LIN {X 0,Y 467.685,Z 587.224,A -85,B 0,C 180,E1 -7551.357,E2 -7551.357} C_VEL
LIN {X 0,Y 467.743,Z 587.223,A -85,B 0,C 180,E1 -7553.963,E2 -7553.963} C_VEL
LIN {X 0,Y 467.864,Z 587.201,A -85,B 0,C 180,E1 -7557.417,E2 -7557.417} C_VEL
LIN {X 0,Y 467.888,Z 587.204,A -85,B 0,C 180,E1 -7560,E2 -7560} C_VEL
LIN {X 0,Y 467.864,Z 587.204,A -85,B 0,C 180,E1 -7562.583,E2 -7562.583} C_VEL
LIN {X 0,Y 467.748,Z 587.22,A -85,B 0,C 180,E1 -7566.037,E2 -7566.037} C_VEL
LIN {X 0,Y 467.686,Z 587.227,A -85,B 0,C 180,E1 -7568.643,E2 -7568.643} C_VEL
LIN {X 0,Y 467.662,Z 587.231,A -85,B 0,C 180,E1 -7572.145,E2 -7572.145} C_VEL
LIN {X 0,Y 467.645,Z 587.228,A -85,B 0,C 180,E1 -7575.695,E2 -7575.695} C_VEL
LIN {X 0,Y 467.619,Z 587.237,A -85,B 0,C 180,E1 -7578.763,E2 -7578.763} C_VEL
LIN {X 0,Y 467.586,Z 587.236,A -85,B 0,C 180,E1 -7581.268,E2 -7581.268} C_VEL
LIN {X 0,Y 467.576,Z 587.237,A -85,B 0,C 180,E1 -7583.943,E2 -7583.943} C_VEL
LIN {X 0,Y 467.622,Z 587.238,A -85,B 0,C 180,E1 -7586.8,E2 -7586.8} C_VEL
LIN {X 0,Y 467.56,Z 587.238,A -85,B 0,C 180,E1 -7589.738,E2 -7589.738} C_VEL
LIN {X 0,Y 467.589,Z 587.243,A -85,B 0,C 180,E1 -7592.758,E2 -7592.758} C_VEL
LIN {X 0,Y 467.559,Z 587.238,A -85,B 0,C 180,E1 -7595.889,E2 -7595.889} C_VEL
LIN {X 0,Y 467.581,Z 587.241,A -85,B 0,C 180,E1 -7599.145,E2 -7599.145} C_VEL
LIN {X 0,Y 467.592,Z 587.238,A -85,B 0,C 180,E1 -7602.567,E2 -7602.567} C_VEL
LIN {X 0,Y 467.576,Z 587.245,A -85,B 0,C 180,E1 -7605.053,E2 -7605.053} C_VEL
LIN {X 0,Y 467.594,Z 587.238,A -85,B 0,C 180,E1 -7607.44,E2 -7607.44} C_VEL
LIN {X 0,Y 467.588,Z 587.24,A -85,B 0,C 180,E1 -7610.855,E2 -7610.855} C_VEL
LIN {X 0,Y 467.565,Z 587.238,A -85,B 0,C 180,E1 -7614.26,E2 -7614.26} C_VEL
LIN {X 0,Y 467.587,Z 587.243,A -85,B 0,C 180,E1 -7617.32,E2 -7617.32} C_VEL
LIN {X 0,Y 467.574,Z 587.241,A -85,B 0,C 180,E1 -7620.667,E2 -7620.667} C_VEL
LIN {X 0,Y 467.688,Z 587.373,A -85,B 0,C 180,E1 -7622.729,E2 -7622.729} C_VEL
LIN {X 0,Y 470.217,Z 599.912,A -85,B 0,C 180,E1 -7625.024,E2 -7625.024} C_VEL
LIN {X 0,Y 470.285,Z 605.726,A -85,B 0,C 180,E1 -7626.017,E2 -7626.017} C_VEL
LIN {X 0,Y 469.404,Z 623.346,A -85,B 0,C 180,E1 -7628.94,E2 -7628.94} C_VEL
LIN {X 0,Y 468.7,Z 641.213,A -85,B 0,C 180,E1 -7631.871,E2 -7631.871} C_VEL
LIN {X 0,Y 468.432,Z 648.08,A -85,B 0,C 180,E1 -7632.987,E2 -7632.987} C_VEL
LIN {X 0,Y 471.155,Z 668.22,A -85,B 0,C 180,E1 -7633.412,E2 -7633.412} C_VEL
LIN {X 0,Y 470.414,Z 757.203,A -85,B 0,C 180,E1 -7634.843,E2 -7634.843} C_VEL
LIN {X 0,Y 469.976,Z 771.033,A -85,B 0,C 180,E1 -7635.244,E2 -7635.244} C_VEL
LIN {X 0,Y 469.566,Z 784.014,A -85,B 0,C 180,E1 -7635.812,E2 -7635.812} C_VEL
LIN {X 0,Y 469.023,Z 796.625,A -85,B 0,C 180,E1 -7636.569,E2 -7636.569} C_VEL
LIN {X 0,Y 468.588,Z 807.32,A -85,B 0,C 180,E1 -7637.39,E2 -7637.39} C_VEL
LIN {X 0,Y 468.191,Z 817.018,A -85,B 0,C 180,E1 -7638.307,E2 -7638.307} C_VEL
LIN {X 0,Y 467.667,Z 826.375,A -85,B 0,C 180,E1 -7639.391,E2 -7639.391} C_VEL
LIN {X 0,Y 467.284,Z 835.456,A -85,B 0,C 180,E1 -7640.695,E2 -7640.695} C_VEL
LIN {X 0,Y 467.022,Z 842.773,A -85,B 0,C 180,E1 -7641.998,E2 -7641.998} C_VEL
LIN {X 0,Y 466.855,Z 847.713,A -85,B 0,C 180,E1 -7643.082,E2 -7643.082} C_VEL
LIN {X 0,Y 466.787,Z 852.513,A -85,B 0,C 180,E1 -7644.383,E2 -7644.383} C_VEL
LIN {X 0,Y 466.666,Z 856.175,A -85,B 0,C 180,E1 -7645.681,E2 -7645.681} C_VEL
LIN {X 0,Y 466.728,Z 858.07,A -85,B 0,C 180,E1 -7646.546,E2 -7646.546} C_VEL
LIN {X 0,Y 466.7,Z 859.486,A -85,B 0,C 180,E1 -7647.41,E2 -7647.41} C_VEL
LIN {X 0,Y 466.693,Z 860.49,A -85,B 0,C 180,E1 -7648.273,E2 -7648.273} C_VEL
LIN {X 0,Y 466.598,Z 861.304,A -85,B 0,C 180,E1 -7649.999,E2 -7649.999} C_VEL
LIN {X 0,Y 466.62,Z 861.075,A -85,B 0,C 180,E1 -7650.862,E2 -7650.862} C_VEL
LIN {X 0,Y 466.694,Z 860.447,A -85,B 0,C 180,E1 -7651.725,E2 -7651.725} C_VEL
LIN {X 0,Y 466.71,Z 859.42,A -85,B 0,C 180,E1 -7652.588,E2 -7652.588} C_VEL
LIN {X 0,Y 466.728,Z 857.982,A -85,B 0,C 180,E1 -7653.452,E2 -7653.452} C_VEL
LIN {X 0,Y 466.7,Z 854.965,A -85,B 0,C 180,E1 -7654.75,E2 -7654.75} C_VEL
LIN {X 0,Y 466.768,Z 850.892,A -85,B 0,C 180,E1 -7656.049,E2 -7656.049} C_VEL
LIN {X 0,Y 466.928,Z 844.629,A -85,B 0,C 180,E1 -7657.567,E2 -7657.567} C_VEL
LIN {X 0,Y 467.165,Z 837.801,A -85,B 0,C 180,E1 -7658.869,E2 -7658.869} C_VEL
LIN {X 0,Y 467.497,Z 829.332,A -85,B 0,C 180,E1 -7660.173,E2 -7660.173} C_VEL
LIN {X 0,Y 467.921,Z 820.622,A -85,B 0,C 180,E1 -7661.259,E2 -7661.259} C_VEL
LIN {X 0,Y 468.377,Z 810.405,A -85,B 0,C 180,E1 -7662.298,E2 -7662.298} C_VEL
LIN {X 0,Y 468.893,Z 799.253,A -85,B 0,C 180,E1 -7663.212,E2 -7663.212} C_VEL
LIN {X 0,Y 469.367,Z 787.483,A -85,B 0,C 180,E1 -7663.971,E2 -7663.971} C_VEL
LIN {X 0,Y 469.795,Z 775.278,A -85,B 0,C 180,E1 -7664.566,E2 -7664.566} C_VEL
LIN {X 0,Y 470.222,Z 762.96,A -85,B 0,C 180,E1 -7664.995,E2 -7664.995} C_VEL
LIN {X 0,Y 470.484,Z 749.275,A -85,B 0,C 180,E1 -7665.291,E2 -7665.291} C_VEL
LIN {X 0,Y 471.087,Z 666.51,A -85,B 0,C 180,E1 -7666.607,E2 -7666.607} C_VEL
LIN {X 0,Y 468.342,Z 647.034,A -85,B 0,C 180,E1 -7667.056,E2 -7667.056} C_VEL
LIN {X 0,Y 469.089,Z 627.979,A -85,B 0,C 180,E1 -7670.156,E2 -7670.156} C_VEL
LIN {X 0,Y 469.848,Z 610.048,A -85,B 0,C 180,E1 -7673.118,E2 -7673.118} C_VEL
LIN {X 0,Y 470.271,Z 600.433,A -85,B 0,C 180,E1 -7674.735,E2 -7674.735} C_VEL
LIN {X 0,Y 467.669,Z 587.232,A -85,B 0,C 180,E1 -7677.189,E2 -7677.189} C_VEL
LIN {X 0,Y 467.568,Z 587.248,A -85,B 0,C 180,E1 -7680.733,E2 -7680.733} C_VEL
LIN {X 0,Y 467.584,Z 587.24,A -85,B 0,C 180,E1 -7683.787,E2 -7683.787} C_VEL
LIN {X 0,Y 467.548,Z 587.244,A -85,B 0,C 180,E1 -7687.186,E2 -7687.186} C_VEL
LIN {X 0,Y 467.591,Z 587.243,A -85,B 0,C 180,E1 -7690.262,E2 -7690.262} C_VEL
LIN {X 0,Y 467.582,Z 587.245,A -85,B 0,C 180,E1 -7692.566,E2 -7692.566} C_VEL
LIN {X 0,Y 467.57,Z 587.245,A -85,B 0,C 180,E1 -7696.175,E2 -7696.175} C_VEL
LIN {X 0,Y 467.584,Z 587.242,A -85,B 0,C 180,E1 -7698.721,E2 -7698.721} C_VEL
LIN {X 0,Y 467.573,Z 587.238,A -85,B 0,C 180,E1 -7701.405,E2 -7701.405} C_VEL
LIN {X 0,Y 467.557,Z 587.244,A -85,B 0,C 180,E1 -7704.259,E2 -7704.259} C_VEL
LIN {X 0,Y 467.576,Z 587.237,A -85,B 0,C 180,E1 -7707.32,E2 -7707.32} C_VEL
LIN {X 0,Y 467.572,Z 587.24,A -85,B 0,C 180,E1 -7710.665,E2 -7710.665} C_VEL
LIN {X 0,Y 467.62,Z 587.231,A -85,B 0,C 180,E1 -7713.2,E2 -7713.2} C_VEL
LIN {X 0,Y 467.585,Z 587.24,A -85,B 0,C 180,E1 -7716.467,E2 -7716.467} C_VEL
LIN {X 0,Y 467.616,Z 587.232,A -85,B 0,C 180,E1 -7719.777,E2 -7719.777} C_VEL
LIN {X 0,Y 467.601,Z 587.239,A -85,B 0,C 180,E1 -7722.506,E2 -7722.506} C_VEL
LIN {X 0,Y 467.598,Z 587.234,A -85,B 0,C 180,E1 -7725.196,E2 -7725.196} C_VEL
LIN {X 0,Y 467.674,Z 587.227,A -85,B 0,C 180,E1 -7727.855,E2 -7727.855} C_VEL
LIN {X 0,Y 467.674,Z 587.226,A -85,B 0,C 180,E1 -7731.357,E2 -7731.357} C_VEL
LIN {X 0,Y 467.735,Z 587.222,A -85,B 0,C 180,E1 -7733.962,E2 -7733.962} C_VEL
LIN {X 0,Y 467.852,Z 587.204,A -85,B 0,C 180,E1 -7737.417,E2 -7737.417} C_VEL
LIN {X 0,Y 467.874,Z 587.206,A -85,B 0,C 180,E1 -7740,E2 -7740} C_VEL
LIN {X 0,Y 467.852,Z 587.209,A -85,B 0,C 180,E1 -7742.583,E2 -7742.583} C_VEL
LIN {X 0,Y 467.746,Z 587.224,A -85,B 0,C 180,E1 -7746.037,E2 -7746.037} C_VEL
LIN {X 0,Y 467.674,Z 587.231,A -85,B 0,C 180,E1 -7748.643,E2 -7748.643} C_VEL
LIN {X 0,Y 467.675,Z 587.235,A -85,B 0,C 180,E1 -7752.145,E2 -7752.145} C_VEL
LIN {X 0,Y 467.661,Z 587.255,A -85,B 0,C 180,E1 -7755.359,E2 -7755.359} C_VEL
LIN {X 0,Y 468.623,Z 593.879,A -85,B 0,C 180,E1 -7757.004,E2 -7757.004} C_VEL
LIN {X 0,Y 468.56,Z 598.288,A -85,B 0,C 180,E1 -7758.049,E2 -7758.049} C_VEL
LIN {X 0,Y 471.347,Z 611.243,A -85,B 0,C 180,E1 -7758.388,E2 -7758.388} C_VEL
LIN {X 0,Y 470.527,Z 704.015,A -85,B 0,C 180,E1 -7759.891,E2 -7759.891} C_VEL
LIN {X 0,Y 470.243,Z 717.329,A -85,B 0,C 180,E1 -7760.276,E2 -7760.276} C_VEL
LIN {X 0,Y 469.916,Z 729.669,A -85,B 0,C 180,E1 -7760.806,E2 -7760.806} C_VEL
LIN {X 0,Y 469.564,Z 741.214,A -85,B 0,C 180,E1 -7761.474,E2 -7761.474} C_VEL
LIN {X 0,Y 469.048,Z 752.847,A -85,B 0,C 180,E1 -7762.346,E2 -7762.346} C_VEL
LIN {X 0,Y 468.564,Z 762.941,A -85,B 0,C 180,E1 -7763.293,E2 -7763.293} C_VEL
LIN {X 0,Y 468.102,Z 772.4,A -85,B 0,C 180,E1 -7764.386,E2 -7764.386} C_VEL
LIN {X 0,Y 467.651,Z 780.999,A -85,B 0,C 180,E1 -7765.621,E2 -7765.621} C_VEL
LIN {X 0,Y 467.375,Z 787.765,A -85,B 0,C 180,E1 -7766.815,E2 -7766.815} C_VEL
LIN {X 0,Y 467.121,Z 794.44,A -85,B 0,C 180,E1 -7768.29,E2 -7768.29} C_VEL
LIN {X 0,Y 466.865,Z 799.568,A -85,B 0,C 180,E1 -7769.786,E2 -7769.786} C_VEL
LIN {X 0,Y 466.807,Z 802.45,A -85,B 0,C 180,E1 -7770.892,E2 -7770.892} C_VEL
LIN {X 0,Y 466.639,Z 805.331,A -85,B 0,C 180,E1 -7772.5,E2 -7772.5} C_VEL
LIN {X 0,Y 466.576,Z 806.772,A -85,B 0,C 180,E1 -7774.061,E2 -7774.061} C_VEL
LIN {X 0,Y 466.56,Z 806.938,A -85,B 0,C 180,E1 -7775.57,E2 -7775.57} C_VEL
LIN {X 0,Y 466.592,Z 805.927,A -85,B 0,C 180,E1 -7777.049,E2 -7777.049} C_VEL
LIN {X 0,Y 466.696,Z 803.852,A -85,B 0,C 180,E1 -7778.459,E2 -7778.459} C_VEL
LIN {X 0,Y 466.821,Z 800.709,A -85,B 0,C 180,E1 -7779.845,E2 -7779.845} C_VEL
LIN {X 0,Y 467.007,Z 795.499,A -85,B 0,C 180,E1 -7781.465,E2 -7781.465} C_VEL
LIN {X 0,Y 467.231,Z 789.418,A -85,B 0,C 180,E1 -7782.894,E2 -7782.894} C_VEL
LIN {X 0,Y 467.618,Z 781.516,A -85,B 0,C 180,E1 -7784.335,E2 -7784.335} C_VEL
LIN {X 0,Y 468.027,Z 773.201,A -85,B 0,C 180,E1 -7785.55,E2 -7785.55} C_VEL
LIN {X 0,Y 468.454,Z 764.065,A -85,B 0,C 180,E1 -7786.639,E2 -7786.639} C_VEL
LIN {X 0,Y 468.921,Z 754.232,A -85,B 0,C 180,E1 -7787.591,E2 -7787.591} C_VEL
LIN {X 0,Y 469.398,Z 742.869,A -85,B 0,C 180,E1 -7788.471,E2 -7788.471} C_VEL
LIN {X 0,Y 469.882,Z 730.838,A -85,B 0,C 180,E1 -7789.197,E2 -7789.197} C_VEL
LIN {X 0,Y 470.193,Z 717.902,A -85,B 0,C 180,E1 -7789.774,E2 -7789.774} C_VEL
LIN {X 0,Y 470.298,Z 712.356,A -85,B 0,C 180,E1 -7789.964,E2 -7789.964} C_VEL
LIN {X 0,Y 469.848,Z 706.643,A -85,B 0,C 180,E1 -7790.143,E2 -7790.143} C_VEL
LIN {X 0,Y 464.422,Z 688.031,A -85,B 0,C 180,E1 -7790.669,E2 -7790.669} C_VEL
LIN {X 0,Y 463.83,Z 682.219,A -85,B 0,C 180,E1 -7790.78,E2 -7790.78} C_VEL
LIN {X 0,Y 464.42,Z 611.549,A -85,B 0,C 180,E1 -7791.929,E2 -7791.929} C_VEL
LIN {X 0,Y 461.453,Z 597.515,A -85,B 0,C 180,E1 -7792.301,E2 -7792.301} C_VEL
LIN {X 0,Y 461.33,Z 592.208,A -85,B 0,C 180,E1 -7793.551,E2 -7793.551} C_VEL
LIN {X 0,Y 460.592,Z 588.114,A -85,B 0,C 180,E1 -7794.563,E2 -7794.563} C_VEL
LIN {X 0,Y 460.528,Z 588.121,A -85,B 0,C 180,E1 -7797.717,E2 -7797.717} C_VEL
LIN {X 0,Y 460.536,Z 588.114,A -85,B 0,C 180,E1 -7800.77,E2 -7800.77} C_VEL
LIN {X 0,Y 460.56,Z 588.114,A -85,B 0,C 180,E1 -7803.736,E2 -7803.736} C_VEL
LIN {X 0,Y 460.544,Z 588.115,A -85,B 0,C 180,E1 -7806.625,E2 -7806.625} C_VEL
LIN {X 0,Y 460.551,Z 588.112,A -85,B 0,C 180,E1 -7809.454,E2 -7809.454} C_VEL
LIN {X 0,Y 460.559,Z 588.119,A -85,B 0,C 180,E1 -7812.231,E2 -7812.231} C_VEL
LIN {X 0,Y 460.565,Z 588.111,A -85,B 0,C 180,E1 -7814.966,E2 -7814.966} C_VEL
LIN {X 0,Y 460.63,Z 588.103,A -85,B 0,C 180,E1 -7817.667,E2 -7817.667} C_VEL
LIN {X 0,Y 460.629,Z 588.102,A -85,B 0,C 180,E1 -7821.225,E2 -7821.225} C_VEL
LIN {X 0,Y 460.71,Z 588.093,A -85,B 0,C 180,E1 -7823.871,E2 -7823.871} C_VEL
LIN {X 0,Y 460.826,Z 588.077,A -85,B 0,C 180,E1 -7827.379,E2 -7827.379} C_VEL
LIN {X 0,Y 460.854,Z 588.076,A -85,B 0,C 180,E1 -7830.001,E2 -7830.001} C_VEL
LIN {X 0,Y 460.827,Z 588.086,A -85,B 0,C 180,E1 -7832.623,E2 -7832.623} C_VEL
LIN {X 0,Y 460.712,Z 588.093,A -85,B 0,C 180,E1 -7836.131,E2 -7836.131} C_VEL
LIN {X 0,Y 460.632,Z 588.109,A -85,B 0,C 180,E1 -7838.777,E2 -7838.777} C_VEL
LIN {X 0,Y 460.616,Z 588.108,A -85,B 0,C 180,E1 -7842.446,E2 -7842.446} C_VEL
LIN {X 0,Y 460.603,Z 588.105,A -85,B 0,C 180,E1 -7845.998,E2 -7845.998} C_VEL
LIN {X 0,Y 460.574,Z 588.117,A -85,B 0,C 180,E1 -7848.903,E2 -7848.903} C_VEL
LIN {X 0,Y 460.519,Z 588.117,A -85,B 0,C 180,E1 -7851.486,E2 -7851.486} C_VEL
LIN {X 0,Y 460.545,Z 588.113,A -85,B 0,C 180,E1 -7854.333,E2 -7854.333} C_VEL
LIN {X 0,Y 460.577,Z 588.114,A -85,B 0,C 180,E1 -7857.244,E2 -7857.244} C_VEL
LIN {X 0,Y 460.514,Z 588.116,A -85,B 0,C 180,E1 -7860.241,E2 -7860.241} C_VEL
LIN {X 0,Y 460.533,Z 588.12,A -85,B 0,C 180,E1 -7863.325,E2 -7863.325} C_VEL
LIN {X 0,Y 460.481,Z 588.121,A -85,B 0,C 180,E1 -7866.53,E2 -7866.53} C_VEL
LIN {X 0,Y 460.536,Z 588.115,A -85,B 0,C 180,E1 -7869.863,E2 -7869.863} C_VEL
LIN {X 0,Y 460.517,Z 588.119,A -85,B 0,C 180,E1 -7872.901,E2 -7872.901} C_VEL
LIN {X 0,Y 460.513,Z 588.119,A -85,B 0,C 180,E1 -7875.831,E2 -7875.831} C_VEL
LIN {X 0,Y 460.535,Z 588.116,A -85,B 0,C 180,E1 -7878.989,E2 -7878.989} C_VEL
LIN {X 0,Y 460.523,Z 588.121,A -85,B 0,C 180,E1 -7881.267,E2 -7881.267} C_VEL
LIN {X 0,Y 460.515,Z 588.116,A -85,B 0,C 180,E1 -7884.555,E2 -7884.555} C_VEL
LIN {X 0,Y 460.536,Z 588.12,A -85,B 0,C 180,E1 -7887.716,E2 -7887.716} C_VEL
LIN {X 0,Y 460.544,Z 588.112,A -85,B 0,C 180,E1 -7890.769,E2 -7890.769} C_VEL
LIN {X 0,Y 460.561,Z 588.119,A -85,B 0,C 180,E1 -7893.735,E2 -7893.735} C_VEL
LIN {X 0,Y 460.549,Z 588.112,A -85,B 0,C 180,E1 -7896.624,E2 -7896.624} C_VEL
LIN {X 0,Y 460.556,Z 588.115,A -85,B 0,C 180,E1 -7899.453,E2 -7899.453} C_VEL
LIN {X 0,Y 460.555,Z 588.115,A -85,B 0,C 180,E1 -7902.23,E2 -7902.23} C_VEL
LIN {X 0,Y 460.57,Z 588.109,A -85,B 0,C 180,E1 -7904.965,E2 -7904.965} C_VEL
LIN {X 0,Y 460.615,Z 588.105,A -85,B 0,C 180,E1 -7908.559,E2 -7908.559} C_VEL
LIN {X 0,Y 460.701,Z 588.101,A -85,B 0,C 180,E1 -7912.109,E2 -7912.109} C_VEL
LIN {X 0,Y 460.7,Z 588.094,A -85,B 0,C 180,E1 -7914.748,E2 -7914.748} C_VEL
LIN {X 0,Y 460.805,Z 588.08,A -85,B 0,C 180,E1 -7917.378,E2 -7917.378} C_VEL
LIN {X 0,Y 460.858,Z 588.079,A -85,B 0,C 180,E1 -7920,E2 -7920} C_VEL
LIN {X 0,Y 460.805,Z 588.083,A -85,B 0,C 180,E1 -7922.623,E2 -7922.623} C_VEL
LIN {X 0,Y 460.714,Z 588.097,A -85,B 0,C 180,E1 -7926.13,E2 -7926.13} C_VEL
LIN {X 0,Y 460.633,Z 588.104,A -85,B 0,C 180,E1 -7928.776,E2 -7928.776} C_VEL
LIN {X 0,Y 460.619,Z 588.112,A -85,B 0,C 180,E1 -7932.445,E2 -7932.445} C_VEL
LIN {X 0,Y 460.606,Z 588.107,A -85,B 0,C 180,E1 -7935.997,E2 -7935.997} C_VEL
LIN {X 0,Y 460.574,Z 588.109,A -85,B 0,C 180,E1 -7939.615,E2 -7939.615} C_VEL
LIN {X 0,Y 460.517,Z 588.122,A -85,B 0,C 180,E1 -7942.429,E2 -7942.429} C_VEL
LIN {X 0,Y 460.563,Z 588.11,A -85,B 0,C 180,E1 -7945.799,E2 -7945.799} C_VEL
LIN {X 0,Y 460.558,Z 588.113,A -85,B 0,C 180,E1 -7948.233,E2 -7948.233} C_VEL
LIN {X 0,Y 460.526,Z 588.117,A -85,B 0,C 180,E1 -7951.283,E2 -7951.283} C_VEL
LIN {X 0,Y 460.538,Z 588.117,A -85,B 0,C 180,E1 -7954.505,E2 -7954.505} C_VEL
LIN {X 0,Y 460.507,Z 588.118,A -85,B 0,C 180,E1 -7957.623,E2 -7957.623} C_VEL
LIN {X 0,Y 460.544,Z 588.113,A -85,B 0,C 180,E1 -7960.269,E2 -7960.269} C_VEL
LIN {X 0,Y 460.506,Z 588.12,A -85,B 0,C 180,E1 -7963.375,E2 -7963.375} C_VEL
LIN {X 0,Y 460.506,Z 588.12,A -85,B 0,C 180,E1 -7966.624,E2 -7966.624} C_VEL
LIN {X 0,Y 460.547,Z 588.113,A -85,B 0,C 180,E1 -7969.73,E2 -7969.73} C_VEL
LIN {X 0,Y 460.505,Z 588.119,A -85,B 0,C 180,E1 -7972.523,E2 -7972.523} C_VEL
LIN {X 0,Y 460.552,Z 588.117,A -85,B 0,C 180,E1 -7975.623,E2 -7975.623} C_VEL
LIN {X 0,Y 460.542,Z 588.117,A -85,B 0,C 180,E1 -7978.744,E2 -7978.744} C_VEL
LIN {X 0,Y 460.586,Z 588.113,A -85,B 0,C 180,E1 -7982.253,E2 -7982.253} C_VEL
LIN {X 0,Y 460.625,Z 588.289,A -85,B 0,C 180,E1 -7982.51,E2 -7982.51} C_VEL
LIN {X 0,Y 463.403,Z 601.997,A -85,B 0,C 180,E1 -7985.057,E2 -7985.057} C_VEL
LIN {X 0,Y 463.036,Z 613.34,A -85,B 0,C 180,E1 -7986.993,E2 -7986.993} C_VEL
LIN {X 0,Y 462.049,Z 633.966,A -85,B 0,C 180,E1 -7990.449,E2 -7990.449} C_VEL
LIN {X 0,Y 461.432,Z 647.712,A -85,B 0,C 180,E1 -7992.723,E2 -7992.723} C_VEL
LIN {X 0,Y 464.321,Z 668.327,A -85,B 0,C 180,E1 -7993.177,E2 -7993.177} C_VEL
LIN {X 0,Y 463.52,Z 757.447,A -85,B 0,C 180,E1 -7994.64,E2 -7994.64} C_VEL
LIN {X 0,Y 463.053,Z 771.055,A -85,B 0,C 180,E1 -7995.047,E2 -7995.047} C_VEL
LIN {X 0,Y 462.656,Z 783.387,A -85,B 0,C 180,E1 -7995.596,E2 -7995.596} C_VEL
LIN {X 0,Y 462.086,Z 796.048,A -85,B 0,C 180,E1 -7996.364,E2 -7996.364} C_VEL
LIN {X 0,Y 461.58,Z 807.608,A -85,B 0,C 180,E1 -7997.267,E2 -7997.267} C_VEL
LIN {X 0,Y 461.138,Z 817.528,A -85,B 0,C 180,E1 -7998.237,E2 -7998.237} C_VEL
LIN {X 0,Y 460.551,Z 827.532,A -85,B 0,C 180,E1 -7999.448,E2 -7999.448} C_VEL
LIN {X 0,Y 460.192,Z 836.353,A -85,B 0,C 180,E1 -8000.772,E2 -8000.772} C_VEL
LIN {X 0,Y 459.899,Z 843.382,A -85,B 0,C 180,E1 -8002.094,E2 -8002.094} C_VEL
LIN {X 0,Y 459.715,Z 849.579,A -85,B 0,C 180,E1 -8003.568,E2 -8003.568} C_VEL
LIN {X 0,Y 459.631,Z 854.675,A -85,B 0,C 180,E1 -8005.175,E2 -8005.175} C_VEL
LIN {X 0,Y 459.625,Z 857.654,A -85,B 0,C 180,E1 -8006.493,E2 -8006.493} C_VEL
LIN {X 0,Y 459.621,Z 859.074,A -85,B 0,C 180,E1 -8007.37,E2 -8007.37} C_VEL
LIN {X 0,Y 459.63,Z 860.08,A -85,B 0,C 180,E1 -8008.247,E2 -8008.247} C_VEL
LIN {X 0,Y 459.53,Z 860.893,A -85,B 0,C 180,E1 -8009.999,E2 -8009.999} C_VEL
LIN {X 0,Y 459.553,Z 860.662,A -85,B 0,C 180,E1 -8010.875,E2 -8010.875} C_VEL
LIN {X 0,Y 459.631,Z 860.032,A -85,B 0,C 180,E1 -8011.751,E2 -8011.751} C_VEL
LIN {X 0,Y 459.629,Z 859.002,A -85,B 0,C 180,E1 -8012.628,E2 -8012.628} C_VEL
LIN {X 0,Y 459.625,Z 857.558,A -85,B 0,C 180,E1 -8013.506,E2 -8013.506} C_VEL
LIN {X 0,Y 459.631,Z 854.537,A -85,B 0,C 180,E1 -8014.823,E2 -8014.823} C_VEL
LIN {X 0,Y 459.714,Z 849.394,A -85,B 0,C 180,E1 -8016.43,E2 -8016.43} C_VEL
LIN {X 0,Y 459.896,Z 843.15,A -85,B 0,C 180,E1 -8017.904,E2 -8017.904} C_VEL
LIN {X 0,Y 460.188,Z 836.077,A -85,B 0,C 180,E1 -8019.227,E2 -8019.227} C_VEL
LIN {X 0,Y 460.542,Z 827.213,A -85,B 0,C 180,E1 -8020.551,E2 -8020.551} C_VEL
LIN {X 0,Y 461.133,Z 817.155,A -85,B 0,C 180,E1 -8021.761,E2 -8021.761} C_VEL
LIN {X 0,Y 461.538,Z 807.418,A -85,B 0,C 180,E1 -8022.713,E2 -8022.713} C_VEL
LIN {X 0,Y 462.077,Z 795.606,A -85,B 0,C 180,E1 -8023.635,E2 -8023.635} C_VEL
LIN {X 0,Y 462.566,Z 783.903,A -85,B 0,C 180,E1 -8024.349,E2 -8024.349} C_VEL
LIN {X 0,Y 462.97,Z 772.048,A -85,B 0,C 180,E1 -8024.898,E2 -8024.898} C_VEL
LIN {X 0,Y 463.447,Z 759.248,A -85,B 0,C 180,E1 -8025.304,E2 -8025.304} C_VEL
LIN {X 0,Y 463.664,Z 739.802,A -85,B 0,C 180,E1 -8025.663,E2 -8025.663} C_VEL
LIN {X 0,Y 464.286,Z 667.244,A -85,B 0,C 180,E1 -8026.844,E2 -8026.844} C_VEL
LIN {X 0,Y 461.364,Z 646.593,A -85,B 0,C 180,E1 -8027.325,E2 -8027.325} C_VEL
LIN {X 0,Y 462.137,Z 627.591,A -85,B 0,C 180,E1 -8030.472,E2 -8030.472} C_VEL
LIN {X 0,Y 462.992,Z 609.724,A -85,B 0,C 180,E1 -8033.481,E2 -8033.481} C_VEL
LIN {X 0,Y 463.377,Z 602.381,A -85,B 0,C 180,E1 -8034.736,E2 -8034.736} C_VEL
LIN {X 0,Y 461.126,Z 590.452,A -85,B 0,C 180,E1 -8036.962,E2 -8036.962} C_VEL
LIN {X 0,Y 460.623,Z 588.11,A -85,B 0,C 180,E1 -8037.448,E2 -8037.448} C_VEL
LIN {X 0,Y 460.509,Z 588.126,A -85,B 0,C 180,E1 -8040.239,E2 -8040.239} C_VEL
LIN {X 0,Y 460.527,Z 588.119,A -85,B 0,C 180,E1 -8043.324,E2 -8043.324} C_VEL
LIN {X 0,Y 460.476,Z 588.129,A -85,B 0,C 180,E1 -8046.528,E2 -8046.528} C_VEL
LIN {X 0,Y 460.572,Z 588.114,A -85,B 0,C 180,E1 -8049.857,E2 -8049.857} C_VEL
LIN {X 0,Y 460.508,Z 588.124,A -85,B 0,C 180,E1 -8052.899,E2 -8052.899} C_VEL
LIN {X 0,Y 460.519,Z 588.12,A -85,B 0,C 180,E1 -8055.828,E2 -8055.828} C_VEL
LIN {X 0,Y 460.538,Z 588.117,A -85,B 0,C 180,E1 -8058.989,E2 -8058.989} C_VEL
LIN {X 0,Y 460.542,Z 588.114,A -85,B 0,C 180,E1 -8061.268,E2 -8061.268} C_VEL
LIN {X 0,Y 460.507,Z 588.125,A -85,B 0,C 180,E1 -8064.554,E2 -8064.554} C_VEL
LIN {X 0,Y 460.526,Z 588.116,A -85,B 0,C 180,E1 -8067.715,E2 -8067.715} C_VEL
LIN {X 0,Y 460.541,Z 588.114,A -85,B 0,C 180,E1 -8070.769,E2 -8070.769} C_VEL
LIN {X 0,Y 460.561,Z 588.111,A -85,B 0,C 180,E1 -8073.734,E2 -8073.734} C_VEL
LIN {X 0,Y 460.539,Z 588.117,A -85,B 0,C 180,E1 -8076.623,E2 -8076.623} C_VEL
LIN {X 0,Y 460.544,Z 588.112,A -85,B 0,C 180,E1 -8079.452,E2 -8079.452} C_VEL
LIN {X 0,Y 460.552,Z 588.118,A -85,B 0,C 180,E1 -8082.23,E2 -8082.23} C_VEL
LIN {X 0,Y 460.557,Z 588.112,A -85,B 0,C 180,E1 -8084.964,E2 -8084.964} C_VEL
LIN {X 0,Y 460.621,Z 588.104,A -85,B 0,C 180,E1 -8087.666,E2 -8087.666} C_VEL
LIN {X 0,Y 460.621,Z 588.105,A -85,B 0,C 180,E1 -8091.224,E2 -8091.224} C_VEL
LIN {X 0,Y 460.702,Z 588.097,A -85,B 0,C 180,E1 -8093.87,E2 -8093.87} C_VEL
LIN {X 0,Y 460.817,Z 588.08,A -85,B 0,C 180,E1 -8097.377,E2 -8097.377} C_VEL
LIN {X 0,Y 460.845,Z 588.081,A -85,B 0,C 180,E1 -8100,E2 -8100} C_VEL
LIN {X 0,Y 460.817,Z 588.085,A -85,B 0,C 180,E1 -8102.622,E2 -8102.622} C_VEL
LIN {X 0,Y 460.71,Z 588.101,A -85,B 0,C 180,E1 -8106.13,E2 -8106.13} C_VEL
LIN {X 0,Y 460.621,Z 588.109,A -85,B 0,C 180,E1 -8108.776,E2 -8108.776} C_VEL
LIN {X 0,Y 460.621,Z 588.113,A -85,B 0,C 180,E1 -8112.455,E2 -8112.455} C_VEL
LIN {X 0,Y 460.604,Z 588.151,A -85,B 0,C 180,E1 -8115.147,E2 -8115.147} C_VEL
LIN {X 0,Y 461.658,Z 594.738,A -85,B 0,C 180,E1 -8116.813,E2 -8116.813} C_VEL
LIN {X 0,Y 461.637,Z 598.763,A -85,B 0,C 180,E1 -8117.784,E2 -8117.784} C_VEL
LIN {X 0,Y 464.649,Z 612.616,A -85,B 0,C 180,E1 -8118.149,E2 -8118.149} C_VEL
LIN {X 0,Y 463.701,Z 705.035,A -85,B 0,C 180,E1 -8119.68,E2 -8119.68} C_VEL
LIN {X 0,Y 463.395,Z 718.214,A -85,B 0,C 180,E1 -8120.073,E2 -8120.073} C_VEL
LIN {X 0,Y 463.056,Z 730.303,A -85,B 0,C 180,E1 -8120.605,E2 -8120.605} C_VEL
LIN {X 0,Y 462.671,Z 741.501,A -85,B 0,C 180,E1 -8121.264,E2 -8121.264} C_VEL
LIN {X 0,Y 462.181,Z 752.56,A -85,B 0,C 180,E1 -8122.099,E2 -8122.099} C_VEL
LIN {X 0,Y 461.643,Z 762.988,A -85,B 0,C 180,E1 -8123.08,E2 -8123.08} C_VEL
LIN {X 0,Y 461.179,Z 771.492,A -85,B 0,C 180,E1 -8124.059,E2 -8124.059} C_VEL
LIN {X 0,Y 460.725,Z 780.225,A -85,B 0,C 180,E1 -8125.285,E2 -8125.285} C_VEL
LIN {X 0,Y 460.42,Z 787.311,A -85,B 0,C 180,E1 -8126.518,E2 -8126.518} C_VEL
LIN {X 0,Y 460.104,Z 793.769,A -85,B 0,C 180,E1 -8127.919,E2 -8127.919} C_VEL
LIN {X 0,Y 459.873,Z 799.124,A -85,B 0,C 180,E1 -8129.416,E2 -8129.416} C_VEL
LIN {X 0,Y 459.801,Z 801.585,A -85,B 0,C 180,E1 -8130.292,E2 -8130.292} C_VEL
LIN {X 0,Y 459.666,Z 803.882,A -85,B 0,C 180,E1 -8131.321,E2 -8131.321} C_VEL
LIN {X 0,Y 459.574,Z 806.108,A -85,B 0,C 180,E1 -8132.748,E2 -8132.748} C_VEL
LIN {X 0,Y 459.485,Z 807.365,A -85,B 0,C 180,E1 -8134.467,E2 -8134.467} C_VEL
LIN {X 0,Y 459.496,Z 807.26,A -85,B 0,C 180,E1 -8135.844,E2 -8135.844} C_VEL
LIN {X 0,Y 459.506,Z 806.051,A -85,B 0,C 180,E1 -8137.316,E2 -8137.316} C_VEL
LIN {X 0,Y 459.641,Z 803.624,A -85,B 0,C 180,E1 -8138.822,E2 -8138.822} C_VEL
LIN {X 0,Y 459.79,Z 800.407,A -85,B 0,C 180,E1 -8140.161,E2 -8140.161} C_VEL
LIN {X 0,Y 459.94,Z 796.021,A -85,B 0,C 180,E1 -8141.521,E2 -8141.521} C_VEL
LIN {X 0,Y 460.217,Z 789.404,A -85,B 0,C 180,E1 -8143.092,E2 -8143.092} C_VEL
LIN {X 0,Y 460.587,Z 782.691,A -85,B 0,C 180,E1 -8144.339,E2 -8144.339} C_VEL
LIN {X 0,Y 460.994,Z 774.509,A -85,B 0,C 180,E1 -8145.574,E2 -8145.574} C_VEL
LIN {X 0,Y 461.456,Z 765.032,A -85,B 0,C 180,E1 -8146.738,E2 -8146.738} C_VEL
LIN {X 0,Y 461.983,Z 754.509,A -85,B 0,C 180,E1 -8147.779,E2 -8147.779} C_VEL
LIN {X 0,Y 462.517,Z 742.775,A -85,B 0,C 180,E1 -8148.695,E2 -8148.695} C_VEL
LIN {X 0,Y 462.964,Z 731.613,A -85,B 0,C 180,E1 -8149.378,E2 -8149.378} C_VEL
LIN {X 0,Y 463.315,Z 718.787,A -85,B 0,C 180,E1 -8149.966,E2 -8149.966} C_VEL
LIN {X 0,Y 463.6,Z 705.455,A -85,B 0,C 180,E1 -8150.377,E2 -8150.377} C_VEL
LIN {X 0,Y 463.83,Z 682.219,A -85,B 0,C 180,E1 -8150.78,E2 -8150.78} C_VEL
LIN {X 0,Y 463.275,Z 676.413,A -85,B 0,C 180,E1 -8150.894,E2 -8150.894} C_VEL
LIN {X 0,Y 457.987,Z 657.715,A -85,B 0,C 180,E1 -8151.392,E2 -8151.392} C_VEL
LIN {X 0,Y 457.351,Z 651.911,A -85,B 0,C 180,E1 -8151.512,E2 -8151.512} C_VEL
LIN {X 0,Y 457.595,Z 612.095,A -85,B 0,C 180,E1 -8152.176,E2 -8152.176} C_VEL
LIN {X 0,Y 454.518,Z 597.884,A -85,B 0,C 180,E1 -8152.564,E2 -8152.564} C_VEL
LIN {X 0,Y 454.39,Z 593.766,A -85,B 0,C 180,E1 -8153.541,E2 -8153.541} C_VEL
LIN {X 0,Y 453.533,Z 588.993,A -85,B 0,C 180,E1 -8154.745,E2 -8154.745} C_VEL
LIN {X 0,Y 453.46,Z 589.001,A -85,B 0,C 180,E1 -8158.202,E2 -8158.202} C_VEL
LIN {X 0,Y 453.507,Z 588.99,A -85,B 0,C 180,E1 -8161.289,E2 -8161.289} C_VEL
LIN {X 0,Y 453.522,Z 588.993,A -85,B 0,C 180,E1 -8164.286,E2 -8164.286} C_VEL
LIN {X 0,Y 453.479,Z 588.993,A -85,B 0,C 180,E1 -8167.205,E2 -8167.205} C_VEL
LIN {X 0,Y 453.504,Z 588.996,A -85,B 0,C 180,E1 -8170.067,E2 -8170.067} C_VEL
LIN {X 0,Y 453.506,Z 588.99,A -85,B 0,C 180,E1 -8172.877,E2 -8172.877} C_VEL
LIN {X 0,Y 453.513,Z 588.989,A -85,B 0,C 180,E1 -8175.645,E2 -8175.645} C_VEL
LIN {X 0,Y 453.578,Z 588.988,A -85,B 0,C 180,E1 -8178.381,E2 -8178.381} C_VEL
LIN {X 0,Y 453.652,Z 588.974,A -85,B 0,C 180,E1 -8181.986,E2 -8181.986} C_VEL
LIN {X 0,Y 453.672,Z 588.974,A -85,B 0,C 180,E1 -8184.668,E2 -8184.668} C_VEL
LIN {X 0,Y 453.767,Z 588.957,A -85,B 0,C 180,E1 -8187.338,E2 -8187.338} C_VEL
LIN {X 0,Y 453.824,Z 588.951,A -85,B 0,C 180,E1 -8190.001,E2 -8190.001} C_VEL
LIN {X 0,Y 453.767,Z 588.964,A -85,B 0,C 180,E1 -8192.664,E2 -8192.664} C_VEL
LIN {X 0,Y 453.68,Z 588.97,A -85,B 0,C 180,E1 -8196.226,E2 -8196.226} C_VEL
LIN {X 0,Y 453.595,Z 588.984,A -85,B 0,C 180,E1 -8198.914,E2 -8198.914} C_VEL
LIN {X 0,Y 453.566,Z 588.987,A -85,B 0,C 180,E1 -8202.53,E2 -8202.53} C_VEL
LIN {X 0,Y 453.548,Z 588.985,A -85,B 0,C 180,E1 -8206.197,E2 -8206.197} C_VEL
LIN {X 0,Y 453.523,Z 588.993,A -85,B 0,C 180,E1 -8209.041,E2 -8209.041} C_VEL
LIN {X 0,Y 453.48,Z 588.993,A -85,B 0,C 180,E1 -8211.837,E2 -8211.837} C_VEL
LIN {X 0,Y 453.517,Z 588.993,A -85,B 0,C 180,E1 -8214.735,E2 -8214.735} C_VEL
LIN {X 0,Y 453.536,Z 588.986,A -85,B 0,C 180,E1 -8217.96,E2 -8217.96} C_VEL
LIN {X 0,Y 453.469,Z 588.997,A -85,B 0,C 180,E1 -8221.526,E2 -8221.526} C_VEL
LIN {X 0,Y 453.492,Z 588.994,A -85,B 0,C 180,E1 -8224.778,E2 -8224.778} C_VEL
LIN {X 0,Y 453.469,Z 588.994,A -85,B 0,C 180,E1 -8228.312,E2 -8228.312} C_VEL
LIN {X 0,Y 453.498,Z 588.991,A -85,B 0,C 180,E1 -8230.609,E2 -8230.609} C_VEL
LIN {X 0,Y 453.459,Z 589.002,A -85,B 0,C 180,E1 -8233.245,E2 -8233.245} C_VEL
LIN {X 0,Y 453.467,Z 588.997,A -85,B 0,C 180,E1 -8235.779,E2 -8235.779} C_VEL
LIN {X 0,Y 453.483,Z 588.992,A -85,B 0,C 180,E1 -8238.21,E2 -8238.21} C_VEL
LIN {X 0,Y 453.491,Z 588.992,A -85,B 0,C 180,E1 -8240.795,E2 -8240.795} C_VEL
LIN {X 0,Y 453.459,Z 588.998,A -85,B 0,C 180,E1 -8243.918,E2 -8243.918} C_VEL
LIN {X 0,Y 453.487,Z 588.994,A -85,B 0,C 180,E1 -8247.152,E2 -8247.152} C_VEL
LIN {X 0,Y 453.479,Z 588.994,A -85,B 0,C 180,E1 -8250.269,E2 -8250.269} C_VEL
LIN {X 0,Y 453.507,Z 588.992,A -85,B 0,C 180,E1 -8253.294,E2 -8253.294} C_VEL
LIN {X 0,Y 453.502,Z 588.992,A -85,B 0,C 180,E1 -8256.239,E2 -8256.239} C_VEL
LIN {X 0,Y 453.487,Z 588.992,A -85,B 0,C 180,E1 -8259.118,E2 -8259.118} C_VEL
LIN {X 0,Y 453.509,Z 588.996,A -85,B 0,C 180,E1 -8261.945,E2 -8261.945} C_VEL
LIN {X 0,Y 453.545,Z 588.985,A -85,B 0,C 180,E1 -8264.727,E2 -8264.727} C_VEL
LIN {X 0,Y 453.564,Z 588.985,A -85,B 0,C 180,E1 -8268.379,E2 -8268.379} C_VEL
LIN {X 0,Y 453.657,Z 588.978,A -85,B 0,C 180,E1 -8271.985,E2 -8271.985} C_VEL
LIN {X 0,Y 453.674,Z 588.97,A -85,B 0,C 180,E1 -8274.667,E2 -8274.667} C_VEL
LIN {X 0,Y 453.749,Z 588.959,A -85,B 0,C 180,E1 -8277.337,E2 -8277.337} C_VEL
LIN {X 0,Y 453.828,Z 588.955,A -85,B 0,C 180,E1 -8280,E2 -8280} C_VEL
LIN {X 0,Y 453.749,Z 588.962,A -85,B 0,C 180,E1 -8282.663,E2 -8282.663} C_VEL
LIN {X 0,Y 453.682,Z 588.975,A -85,B 0,C 180,E1 -8286.225,E2 -8286.225} C_VEL
LIN {X 0,Y 453.596,Z 588.98,A -85,B 0,C 180,E1 -8288.913,E2 -8288.913} C_VEL
LIN {X 0,Y 453.569,Z 588.988,A -85,B 0,C 180,E1 -8292.529,E2 -8292.529} C_VEL
LIN {X 0,Y 453.55,Z 588.988,A -85,B 0,C 180,E1 -8296.196,E2 -8296.196} C_VEL
LIN {X 0,Y 453.523,Z 588.989,A -85,B 0,C 180,E1 -8299.039,E2 -8299.039} C_VEL
LIN {X 0,Y 453.482,Z 588.993,A -85,B 0,C 180,E1 -8301.836,E2 -8301.836} C_VEL
LIN {X 0,Y 453.513,Z 588.996,A -85,B 0,C 180,E1 -8304.735,E2 -8304.735} C_VEL
LIN {X 0,Y 453.538,Z 588.986,A -85,B 0,C 180,E1 -8307.959,E2 -8307.959} C_VEL
LIN {X 0,Y 453.471,Z 588.994,A -85,B 0,C 180,E1 -8311.525,E2 -8311.525} C_VEL
LIN {X 0,Y 453.493,Z 588.999,A -85,B 0,C 180,E1 -8314.777,E2 -8314.777} C_VEL
LIN {X 0,Y 453.469,Z 588.995,A -85,B 0,C 180,E1 -8318.311,E2 -8318.311} C_VEL
LIN {X 0,Y 453.499,Z 588.994,A -85,B 0,C 180,E1 -8320.609,E2 -8320.609} C_VEL
LIN {X 0,Y 453.462,Z 589,A -85,B 0,C 180,E1 -8323.244,E2 -8323.244} C_VEL
LIN {X 0,Y 453.472,Z 588.994,A -85,B 0,C 180,E1 -8325.779,E2 -8325.779} C_VEL
LIN {X 0,Y 453.484,Z 588.992,A -85,B 0,C 180,E1 -8328.209,E2 -8328.209} C_VEL
LIN {X 0,Y 453.5,Z 588.994,A -85,B 0,C 180,E1 -8330.793,E2 -8330.793} C_VEL
LIN {X 0,Y 453.46,Z 588.996,A -85,B 0,C 180,E1 -8333.917,E2 -8333.917} C_VEL
LIN {X 0,Y 453.488,Z 589,A -85,B 0,C 180,E1 -8337.151,E2 -8337.151} C_VEL
LIN {X 0,Y 453.48,Z 588.996,A -85,B 0,C 180,E1 -8340.268,E2 -8340.268} C_VEL
LIN {X 0,Y 453.55,Z 589.053,A -85,B 0,C 180,E1 -8342.255,E2 -8342.255} C_VEL
LIN {X 0,Y 456.227,Z 601.97,A -85,B 0,C 180,E1 -8344.704,E2 -8344.704} C_VEL
LIN {X 0,Y 456.496,Z 606.053,A -85,B 0,C 180,E1 -8345.437,E2 -8345.437} C_VEL
LIN {X 0,Y 455.641,Z 622.573,A -85,B 0,C 180,E1 -8348.272,E2 -8348.272} C_VEL
LIN {X 0,Y 454.751,Z 640.443,A -85,B 0,C 180,E1 -8351.295,E2 -8351.295} C_VEL
LIN {X 0,Y 454.483,Z 647.394,A -85,B 0,C 180,E1 -8352.464,E2 -8352.464} C_VEL
LIN {X 0,Y 457.498,Z 668.695,A -85,B 0,C 180,E1 -8352.939,E2 -8352.939} C_VEL
LIN {X 0,Y 456.644,Z 756.56,A -85,B 0,C 180,E1 -8354.403,E2 -8354.403} C_VEL
LIN {X 0,Y 456.155,Z 770.316,A -85,B 0,C 180,E1 -8354.815,E2 -8354.815} C_VEL
LIN {X 0,Y 455.76,Z 782.755,A -85,B 0,C 180,E1 -8355.373,E2 -8355.373} C_VEL
LIN {X 0,Y 455.205,Z 793.879,A -85,B 0,C 180,E1 -8356.04,E2 -8356.04} C_VEL
LIN {X 0,Y 454.637,Z 805.78,A -85,B 0,C 180,E1 -8356.957,E2 -8356.957} C_VEL
LIN {X 0,Y 454.2,Z 815.983,A -85,B 0,C 180,E1 -8357.942,E2 -8357.942} C_VEL
LIN {X 0,Y 453.642,Z 825.401,A -85,B 0,C 180,E1 -8359.059,E2 -8359.059} C_VEL
LIN {X 0,Y 453.198,Z 834.519,A -85,B 0,C 180,E1 -8360.403,E2 -8360.403} C_VEL
LIN {X 0,Y 452.879,Z 841.867,A -85,B 0,C 180,E1 -8361.746,E2 -8361.746} C_VEL
LIN {X 0,Y 452.694,Z 846.832,A -85,B 0,C 180,E1 -8362.865,E2 -8362.865} C_VEL
LIN {X 0,Y 452.581,Z 851.652,A -85,B 0,C 180,E1 -8364.206,E2 -8364.206} C_VEL
LIN {X 0,Y 452.503,Z 855.332,A -85,B 0,C 180,E1 -8365.545,E2 -8365.545} C_VEL
LIN {X 0,Y 452.525,Z 857.233,A -85,B 0,C 180,E1 -8366.437,E2 -8366.437} C_VEL
LIN {X 0,Y 452.543,Z 858.659,A -85,B 0,C 180,E1 -8367.329,E2 -8367.329} C_VEL
LIN {X 0,Y 452.538,Z 859.666,A -85,B 0,C 180,E1 -8368.219,E2 -8368.219} C_VEL
LIN {X 0,Y 452.489,Z 860.273,A -85,B 0,C 180,E1 -8369.109,E2 -8369.109} C_VEL
LIN {X 0,Y 452.464,Z 860.482,A -85,B 0,C 180,E1 -8369.999,E2 -8369.999} C_VEL
LIN {X 0,Y 452.489,Z 860.251,A -85,B 0,C 180,E1 -8370.889,E2 -8370.889} C_VEL
LIN {X 0,Y 452.539,Z 859.618,A -85,B 0,C 180,E1 -8371.779,E2 -8371.779} C_VEL
LIN {X 0,Y 452.55,Z 858.584,A -85,B 0,C 180,E1 -8372.669,E2 -8372.669} C_VEL
LIN {X 0,Y 452.525,Z 857.136,A -85,B 0,C 180,E1 -8373.561,E2 -8373.561} C_VEL
LIN {X 0,Y 452.561,Z 854.11,A -85,B 0,C 180,E1 -8374.899,E2 -8374.899} C_VEL
LIN {X 0,Y 452.61,Z 849.459,A -85,B 0,C 180,E1 -8376.395,E2 -8376.395} C_VEL
LIN {X 0,Y 452.782,Z 843.733,A -85,B 0,C 180,E1 -8377.805,E2 -8377.805} C_VEL
LIN {X 0,Y 453.072,Z 836.878,A -85,B 0,C 180,E1 -8379.148,E2 -8379.148} C_VEL
LIN {X 0,Y 453.45,Z 828.377,A -85,B 0,C 180,E1 -8380.492,E2 -8380.492} C_VEL
LIN {X 0,Y 453.953,Z 819.631,A -85,B 0,C 180,E1 -8381.61,E2 -8381.61} C_VEL
LIN {X 0,Y 454.421,Z 809.887,A -85,B 0,C 180,E1 -8382.633,E2 -8382.633} C_VEL
LIN {X 0,Y 454.922,Z 799.646,A -85,B 0,C 180,E1 -8383.512,E2 -8383.512} C_VEL
LIN {X 0,Y 455.459,Z 788.281,A -85,B 0,C 180,E1 -8384.292,E2 -8384.292} C_VEL
LIN {X 0,Y 455.99,Z 775.472,A -85,B 0,C 180,E1 -8384.96,E2 -8384.96} C_VEL
LIN {X 0,Y 456.472,Z 762.726,A -85,B 0,C 180,E1 -8385.429,E2 -8385.429} C_VEL
LIN {X 0,Y 456.76,Z 749.732,A -85,B 0,C 180,E1 -8385.734,E2 -8385.734} C_VEL
LIN {X 0,Y 457.465,Z 667.886,A -85,B 0,C 180,E1 -8387.092,E2 -8387.092} C_VEL
LIN {X 0,Y 454.382,Z 646.269,A -85,B 0,C 180,E1 -8387.589,E2 -8387.589} C_VEL
LIN {X 0,Y 455.227,Z 627.241,A -85,B 0,C 180,E1 -8390.797,E2 -8390.797} C_VEL
LIN {X 0,Y 456.151,Z 609.419,A -85,B 0,C 180,E1 -8393.855,E2 -8393.855} C_VEL
LIN {X 0,Y 456.447,Z 604.49,A -85,B 0,C 180,E1 -8394.71,E2 -8394.71} C_VEL
LIN {X 0,Y 455.36,Z 597.528,A -85,B 0,C 180,E1 -8396.013,E2 -8396.013} C_VEL
LIN {X 0,Y 453.545,Z 588.992,A -85,B 0,C 180,E1 -8397.701,E2 -8397.701} C_VEL
LIN {X 0,Y 453.474,Z 589.004,A -85,B 0,C 180,E1 -8400.758,E2 -8400.758} C_VEL
LIN {X 0,Y 453.475,Z 588.999,A -85,B 0,C 180,E1 -8403.911,E2 -8403.911} C_VEL
LIN {X 0,Y 453.468,Z 588.998,A -85,B 0,C 180,E1 -8407.187,E2 -8407.187} C_VEL
LIN {X 0,Y 453.527,Z 588.991,A -85,B 0,C 180,E1 -8409.444,E2 -8409.444} C_VEL
LIN {X 0,Y 453.458,Z 589.002,A -85,B 0,C 180,E1 -8412.994,E2 -8412.994} C_VEL
LIN {X 0,Y 453.472,Z 588.998,A -85,B 0,C 180,E1 -8415.779,E2 -8415.779} C_VEL
LIN {X 0,Y 453.491,Z 588.999,A -85,B 0,C 180,E1 -8418.21,E2 -8418.21} C_VEL
LIN {X 0,Y 453.527,Z 588.991,A -85,B 0,C 180,E1 -8420.786,E2 -8420.786} C_VEL
LIN {X 0,Y 453.451,Z 588.997,A -85,B 0,C 180,E1 -8423.917,E2 -8423.917} C_VEL
LIN {X 0,Y 453.477,Z 588.995,A -85,B 0,C 180,E1 -8427.15,E2 -8427.15} C_VEL
LIN {X 0,Y 453.507,Z 588.995,A -85,B 0,C 180,E1 -8430.27,E2 -8430.27} C_VEL
LIN {X 0,Y 453.506,Z 588.989,A -85,B 0,C 180,E1 -8433.294,E2 -8433.294} C_VEL
LIN {X 0,Y 453.496,Z 588.996,A -85,B 0,C 180,E1 -8436.238,E2 -8436.238} C_VEL
LIN {X 0,Y 453.475,Z 588.993,A -85,B 0,C 180,E1 -8439.117,E2 -8439.117} C_VEL
LIN {X 0,Y 453.504,Z 588.994,A -85,B 0,C 180,E1 -8441.944,E2 -8441.944} C_VEL
LIN {X 0,Y 453.531,Z 588.989,A -85,B 0,C 180,E1 -8444.726,E2 -8444.726} C_VEL
LIN {X 0,Y 453.593,Z 588.979,A -85,B 0,C 180,E1 -8447.472,E2 -8447.472} C_VEL
LIN {X 0,Y 453.585,Z 588.982,A -85,B 0,C 180,E1 -8451.086,E2 -8451.086} C_VEL
LIN {X 0,Y 453.669,Z 588.973,A -85,B 0,C 180,E1 -8453.774,E2 -8453.774} C_VEL
LIN {X 0,Y 453.758,Z 588.96,A -85,B 0,C 180,E1 -8457.337,E2 -8457.337} C_VEL
LIN {X 0,Y 453.816,Z 588.957,A -85,B 0,C 180,E1 -8460,E2 -8460} C_VEL
LIN {X 0,Y 453.758,Z 588.964,A -85,B 0,C 180,E1 -8462.663,E2 -8462.663} C_VEL
LIN {X 0,Y 453.676,Z 588.977,A -85,B 0,C 180,E1 -8466.225,E2 -8466.225} C_VEL
LIN {X 0,Y 453.585,Z 588.984,A -85,B 0,C 180,E1 -8468.913,E2 -8468.913} C_VEL
LIN {X 0,Y 453.589,Z 588.988,A -85,B 0,C 180,E1 -8472.549,E2 -8472.549} C_VEL
LIN {X 0,Y 453.571,Z 589.101,A -85,B 0,C 180,E1 -8474.928,E2 -8474.928} C_VEL
LIN {X 0,Y 454.689,Z 595.602,A -85,B 0,C 180,E1 -8476.606,E2 -8476.606} C_VEL
LIN {X 0,Y 454.709,Z 599.258,A -85,B 0,C 180,E1 -8477.502,E2 -8477.502} C_VEL
LIN {X 0,Y 457.86,Z 613.374,A -85,B 0,C 180,E1 -8477.889,E2 -8477.889} C_VEL
LIN {X 0,Y 456.869,Z 706.075,A -85,B 0,C 180,E1 -8479.459,E2 -8479.459} C_VEL
LIN {X 0,Y 456.555,Z 719.617,A -85,B 0,C 180,E1 -8479.88,E2 -8479.88} C_VEL
LIN {X 0,Y 456.127,Z 732.171,A -85,B 0,C 180,E1 -8480.458,E2 -8480.458} C_VEL
LIN {X 0,Y 455.652,Z 744.769,A -85,B 0,C 180,E1 -8481.252,E2 -8481.252} C_VEL
LIN {X 0,Y 455.161,Z 755.5,A -85,B 0,C 180,E1 -8482.117,E2 -8482.117} C_VEL
LIN {X 0,Y 454.549,Z 766.374,A -85,B 0,C 180,E1 -8483.22,E2 -8483.22} C_VEL
LIN {X 0,Y 454.07,Z 775.292,A -85,B 0,C 180,E1 -8484.343,E2 -8484.343} C_VEL
LIN {X 0,Y 453.535,Z 784.125,A -85,B 0,C 180,E1 -8485.715,E2 -8485.715} C_VEL
LIN {X 0,Y 453.282,Z 790.569,A -85,B 0,C 180,E1 -8486.969,E2 -8486.969} C_VEL
LIN {X 0,Y 452.987,Z 795.947,A -85,B 0,C 180,E1 -8488.26,E2 -8488.26} C_VEL
LIN {X 0,Y 452.741,Z 800.852,A -85,B 0,C 180,E1 -8489.785,E2 -8489.785} C_VEL
LIN {X 0,Y 452.58,Z 804.463,A -85,B 0,C 180,E1 -8491.344,E2 -8491.344} C_VEL
LIN {X 0,Y 452.484,Z 806.848,A -85,B 0,C 180,E1 -8492.996,E2 -8492.996} C_VEL
LIN {X 0,Y 452.39,Z 807.799,A -85,B 0,C 180,E1 -8494.579,E2 -8494.579} C_VEL
LIN {X 0,Y 452.422,Z 807.489,A -85,B 0,C 180,E1 -8496.178,E2 -8496.178} C_VEL
LIN {X 0,Y 452.457,Z 806.117,A -85,B 0,C 180,E1 -8497.612,E2 -8497.612} C_VEL
LIN {X 0,Y 452.58,Z 803.639,A -85,B 0,C 180,E1 -8499.066,E2 -8499.066} C_VEL
LIN {X 0,Y 452.802,Z 799.523,A -85,B 0,C 180,E1 -8500.684,E2 -8500.684} C_VEL
LIN {X 0,Y 452.964,Z 794.399,A -85,B 0,C 180,E1 -8502.147,E2 -8502.147} C_VEL
LIN {X 0,Y 453.352,Z 787.46,A -85,B 0,C 180,E1 -8503.675,E2 -8503.675} C_VEL
LIN {X 0,Y 453.684,Z 780.203,A -85,B 0,C 180,E1 -8504.948,E2 -8504.948} C_VEL
LIN {X 0,Y 454.238,Z 771.342,A -85,B 0,C 180,E1 -8506.198,E2 -8506.198} C_VEL
LIN {X 0,Y 454.738,Z 761.288,A -85,B 0,C 180,E1 -8507.348,E2 -8507.348} C_VEL
LIN {X 0,Y 455.27,Z 750.569,A -85,B 0,C 180,E1 -8508.334,E2 -8508.334} C_VEL
LIN {X 0,Y 455.809,Z 738.405,A -85,B 0,C 180,E1 -8509.209,E2 -8509.209} C_VEL
LIN {X 0,Y 456.331,Z 725.53,A -85,B 0,C 180,E1 -8509.912,E2 -8509.912} C_VEL
LIN {X 0,Y 456.581,Z 712.383,A -85,B 0,C 180,E1 -8510.42,E2 -8510.42} C_VEL
LIN {X 0,Y 456.901,Z 699.66,A -85,B 0,C 180,E1 -8510.728,E2 -8510.728} C_VEL
LIN {X 0,Y 457.351,Z 651.911,A -85,B 0,C 180,E1 -8511.512,E2 -8511.512} C_VEL
LIN {X 0,Y 456.737,Z 646.113,A -85,B 0,C 180,E1 -8511.632,E2 -8511.632} C_VEL
LIN {X 0,Y 451.527,Z 627.427,A -85,B 0,C 180,E1 -8512.146,E2 -8512.146} C_VEL
LIN {X 0,Y 450.888,Z 621.632,A -85,B 0,C 180,E1 -8512.271,E2 -8512.271} C_VEL
LIN {X 0,Y 450.762,Z 612.94,A -85,B 0,C 180,E1 -8512.426,E2 -8512.426} C_VEL
LIN {X 0,Y 447.56,Z 598.329,A -85,B 0,C 180,E1 -8512.811,E2 -8512.811} C_VEL
LIN {X 0,Y 447.229,Z 593.867,A -85,B 0,C 180,E1 -8513.895,E2 -8513.895} C_VEL
LIN {X 0,Y 446.481,Z 589.871,A -85,B 0,C 180,E1 -8514.937,E2 -8514.937} C_VEL
LIN {X 0,Y 446.415,Z 589.878,A -85,B 0,C 180,E1 -8518.226,E2 -8518.226} C_VEL
LIN {X 0,Y 446.481,Z 589.87,A -85,B 0,C 180,E1 -8521.822,E2 -8521.822} C_VEL
LIN {X 0,Y 446.455,Z 589.868,A -85,B 0,C 180,E1 -8524.849,E2 -8524.849} C_VEL
LIN {X 0,Y 446.446,Z 589.876,A -85,B 0,C 180,E1 -8528.246,E2 -8528.246} C_VEL
LIN {X 0,Y 446.457,Z 589.869,A -85,B 0,C 180,E1 -8531.65,E2 -8531.65} C_VEL
LIN {X 0,Y 446.507,Z 589.866,A -85,B 0,C 180,E1 -8534.481,E2 -8534.481} C_VEL
LIN {X 0,Y 446.539,Z 589.864,A -85,B 0,C 180,E1 -8538.195,E2 -8538.195} C_VEL
LIN {X 0,Y 446.601,Z 589.851,A -85,B 0,C 180,E1 -8541.859,E2 -8541.859} C_VEL
LIN {X 0,Y 446.646,Z 589.85,A -85,B 0,C 180,E1 -8544.584,E2 -8544.584} C_VEL
LIN {X 0,Y 446.711,Z 589.836,A -85,B 0,C 180,E1 -8547.296,E2 -8547.296} C_VEL
LIN {X 0,Y 446.794,Z 589.827,A -85,B 0,C 180,E1 -8550.001,E2 -8550.001} C_VEL
LIN {X 0,Y 446.711,Z 589.843,A -85,B 0,C 180,E1 -8552.706,E2 -8552.706} C_VEL
LIN {X 0,Y 446.649,Z 589.847,A -85,B 0,C 180,E1 -8556.325,E2 -8556.325} C_VEL
LIN {X 0,Y 446.541,Z 589.861,A -85,B 0,C 180,E1 -8559.056,E2 -8559.056} C_VEL
LIN {X 0,Y 446.524,Z 589.867,A -85,B 0,C 180,E1 -8562.731,E2 -8562.731} C_VEL
LIN {X 0,Y 446.499,Z 589.863,A -85,B 0,C 180,E1 -8566.229,E2 -8566.229} C_VEL
LIN {X 0,Y 446.472,Z 589.868,A -85,B 0,C 180,E1 -8569.304,E2 -8569.304} C_VEL
LIN {X 0,Y 446.421,Z 589.872,A -85,B 0,C 180,E1 -8572.2,E2 -8572.2} C_VEL
LIN {X 0,Y 446.461,Z 589.873,A -85,B 0,C 180,E1 -8575.153,E2 -8575.153} C_VEL
LIN {X 0,Y 446.488,Z 589.864,A -85,B 0,C 180,E1 -8578.179,E2 -8578.179} C_VEL
LIN {X 0,Y 446.423,Z 589.873,A -85,B 0,C 180,E1 -8581.776,E2 -8581.776} C_VEL
LIN {X 0,Y 446.433,Z 589.871,A -85,B 0,C 180,E1 -8584.524,E2 -8584.524} C_VEL
LIN {X 0,Y 446.42,Z 589.872,A -85,B 0,C 180,E1 -8588.08,E2 -8588.08} C_VEL
LIN {X 0,Y 446.431,Z 589.874,A -85,B 0,C 180,E1 -8590.918,E2 -8590.918} C_VEL
LIN {X 0,Y 446.404,Z 589.876,A -85,B 0,C 180,E1 -8593.847,E2 -8593.847} C_VEL
LIN {X 0,Y 446.402,Z 589.874,A -85,B 0,C 180,E1 -8596.404,E2 -8596.404} C_VEL
LIN {X 0,Y 446.431,Z 589.874,A -85,B 0,C 180,E1 -8599.083,E2 -8599.083} C_VEL
LIN {X 0,Y 446.412,Z 589.874,A -85,B 0,C 180,E1 -8602.122,E2 -8602.122} C_VEL
LIN {X 0,Y 446.434,Z 589.878,A -85,B 0,C 180,E1 -8605.477,E2 -8605.477} C_VEL
LIN {X 0,Y 446.42,Z 589.872,A -85,B 0,C 180,E1 -8608.7,E2 -8608.7} C_VEL
LIN {X 0,Y 446.49,Z 589.87,A -85,B 0,C 180,E1 -8611.822,E2 -8611.822} C_VEL
LIN {X 0,Y 446.449,Z 589.868,A -85,B 0,C 180,E1 -8614.847,E2 -8614.847} C_VEL
LIN {X 0,Y 446.453,Z 589.87,A -85,B 0,C 180,E1 -8618.245,E2 -8618.245} C_VEL
LIN {X 0,Y 446.457,Z 589.873,A -85,B 0,C 180,E1 -8621.649,E2 -8621.649} C_VEL
LIN {X 0,Y 446.513,Z 589.862,A -85,B 0,C 180,E1 -8624.48,E2 -8624.48} C_VEL
LIN {X 0,Y 446.522,Z 589.865,A -85,B 0,C 180,E1 -8628.193,E2 -8628.193} C_VEL
LIN {X 0,Y 446.606,Z 589.855,A -85,B 0,C 180,E1 -8631.858,E2 -8631.858} C_VEL
LIN {X 0,Y 446.648,Z 589.846,A -85,B 0,C 180,E1 -8634.583,E2 -8634.583} C_VEL
LIN {X 0,Y 446.669,Z 589.849,A -85,B 0,C 180,E1 -8638.197,E2 -8638.197} C_VEL
LIN {X 0,Y 446.798,Z 589.831,A -85,B 0,C 180,E1 -8640,E2 -8640} C_VEL
LIN {X 0,Y 446.696,Z 589.84,A -85,B 0,C 180,E1 -8642.705,E2 -8642.705} C_VEL
LIN {X 0,Y 446.651,Z 589.852,A -85,B 0,C 180,E1 -8646.324,E2 -8646.324} C_VEL
LIN {X 0,Y 446.542,Z 589.857,A -85,B 0,C 180,E1 -8649.055,E2 -8649.055} C_VEL
LIN {X 0,Y 446.527,Z 589.863,A -85,B 0,C 180,E1 -8652.73,E2 -8652.73} C_VEL
LIN {X 0,Y 446.501,Z 589.867,A -85,B 0,C 180,E1 -8656.227,E2 -8656.227} C_VEL
LIN {X 0,Y 446.474,Z 589.866,A -85,B 0,C 180,E1 -8659.303,E2 -8659.303} C_VEL
LIN {X 0,Y 446.424,Z 589.875,A -85,B 0,C 180,E1 -8662.199,E2 -8662.199} C_VEL
LIN {X 0,Y 446.455,Z 589.87,A -85,B 0,C 180,E1 -8665.153,E2 -8665.153} C_VEL
LIN {X 0,Y 446.49,Z 589.865,A -85,B 0,C 180,E1 -8668.178,E2 -8668.178} C_VEL
LIN {X 0,Y 446.425,Z 589.871,A -85,B 0,C 180,E1 -8671.775,E2 -8671.775} C_VEL
LIN {X 0,Y 446.435,Z 589.874,A -85,B 0,C 180,E1 -8674.523,E2 -8674.523} C_VEL
LIN {X 0,Y 446.42,Z 589.872,A -85,B 0,C 180,E1 -8678.079,E2 -8678.079} C_VEL
LIN {X 0,Y 446.433,Z 589.879,A -85,B 0,C 180,E1 -8680.917,E2 -8680.917} C_VEL
LIN {X 0,Y 446.407,Z 589.874,A -85,B 0,C 180,E1 -8683.845,E2 -8683.845} C_VEL
LIN {X 0,Y 446.405,Z 589.875,A -85,B 0,C 180,E1 -8686.403,E2 -8686.403} C_VEL
LIN {X 0,Y 446.433,Z 589.879,A -85,B 0,C 180,E1 -8689.082,E2 -8689.082} C_VEL
LIN {X 0,Y 446.415,Z 589.873,A -85,B 0,C 180,E1 -8692.121,E2 -8692.121} C_VEL
LIN {X 0,Y 446.435,Z 589.877,A -85,B 0,C 180,E1 -8695.477,E2 -8695.477} C_VEL
LIN {X 0,Y 446.421,Z 589.876,A -85,B 0,C 180,E1 -8698.699,E2 -8698.699} C_VEL
LIN {X 0,Y 446.522,Z 590.018,A -85,B 0,C 180,E1 -8702.037,E2 -8702.037} C_VEL
LIN {X 0,Y 449.198,Z 602.859,A -85,B 0,C 180,E1 -8704.515,E2 -8704.515} C_VEL
LIN {X 0,Y 449.609,Z 606.466,A -85,B 0,C 180,E1 -8705.182,E2 -8705.182} C_VEL
LIN {X 0,Y 448.671,Z 623.545,A -85,B 0,C 180,E1 -8708.159,E2 -8708.159} C_VEL
LIN {X 0,Y 447.75,Z 641.39,A -85,B 0,C 180,E1 -8711.229,E2 -8711.229} C_VEL
LIN {X 0,Y 447.488,Z 647,A -85,B 0,C 180,E1 -8712.187,E2 -8712.187} C_VEL
LIN {X 0,Y 450.68,Z 669.634,A -85,B 0,C 180,E1 -8712.703,E2 -8712.703} C_VEL
LIN {X 0,Y 449.774,Z 756.749,A -85,B 0,C 180,E1 -8714.188,E2 -8714.188} C_VEL
LIN {X 0,Y 449.261,Z 770.311,A -85,B 0,C 180,E1 -8714.605,E2 -8714.605} C_VEL
LIN {X 0,Y 448.805,Z 783.14,A -85,B 0,C 180,E1 -8715.199,E2 -8715.199} C_VEL
LIN {X 0,Y 448.194,Z 794.89,A -85,B 0,C 180,E1 -8715.932,E2 -8715.932} C_VEL
LIN {X 0,Y 447.62,Z 806.358,A -85,B 0,C 180,E1 -8716.849,E2 -8716.849} C_VEL
LIN {X 0,Y 447.155,Z 816.514,A -85,B 0,C 180,E1 -8717.864,E2 -8717.864} C_VEL
LIN {X 0,Y 446.528,Z 826.56,A -85,B 0,C 180,E1 -8719.112,E2 -8719.112} C_VEL
LIN {X 0,Y 446.078,Z 835.418,A -85,B 0,C 180,E1 -8720.477,E2 -8720.477} C_VEL
LIN {X 0,Y 445.776,Z 842.483,A -85,B 0,C 180,E1 -8721.842,E2 -8721.842} C_VEL
LIN {X 0,Y 445.555,Z 848.297,A -85,B 0,C 180,E1 -8723.25,E2 -8723.25} C_VEL
LIN {X 0,Y 445.506,Z 852.571,A -85,B 0,C 180,E1 -8724.568,E2 -8724.568} C_VEL
LIN {X 0,Y 445.428,Z 854.908,A -85,B 0,C 180,E1 -8725.474,E2 -8725.474} C_VEL
LIN {X 0,Y 445.426,Z 856.812,A -85,B 0,C 180,E1 -8726.381,E2 -8726.381} C_VEL
LIN {X 0,Y 445.467,Z 858.244,A -85,B 0,C 180,E1 -8727.286,E2 -8727.286} C_VEL
LIN {X 0,Y 445.45,Z 859.252,A -85,B 0,C 180,E1 -8728.191,E2 -8728.191} C_VEL
LIN {X 0,Y 445.427,Z 859.861,A -85,B 0,C 180,E1 -8729.095,E2 -8729.095} C_VEL
LIN {X 0,Y 445.399,Z 860.071,A -85,B 0,C 180,E1 -8729.999,E2 -8729.999} C_VEL
LIN {X 0,Y 445.427,Z 859.84,A -85,B 0,C 180,E1 -8730.903,E2 -8730.903} C_VEL
LIN {X 0,Y 445.452,Z 859.203,A -85,B 0,C 180,E1 -8731.807,E2 -8731.807} C_VEL
LIN {X 0,Y 445.473,Z 858.167,A -85,B 0,C 180,E1 -8732.712,E2 -8732.712} C_VEL
LIN {X 0,Y 445.426,Z 856.715,A -85,B 0,C 180,E1 -8733.617,E2 -8733.617} C_VEL
LIN {X 0,Y 445.492,Z 853.684,A -85,B 0,C 180,E1 -8734.977,E2 -8734.977} C_VEL
LIN {X 0,Y 445.556,Z 848.105,A -85,B 0,C 180,E1 -8736.748,E2 -8736.748} C_VEL
LIN {X 0,Y 445.77,Z 842.251,A -85,B 0,C 180,E1 -8738.156,E2 -8738.156} C_VEL
LIN {X 0,Y 446.066,Z 835.161,A -85,B 0,C 180,E1 -8739.521,E2 -8739.521} C_VEL
LIN {X 0,Y 446.513,Z 826.283,A -85,B 0,C 180,E1 -8740.886,E2 -8740.886} C_VEL
LIN {X 0,Y 447.089,Z 816.209,A -85,B 0,C 180,E1 -8742.136,E2 -8742.136} C_VEL
LIN {X 0,Y 447.573,Z 806.373,A -85,B 0,C 180,E1 -8743.125,E2 -8743.125} C_VEL
LIN {X 0,Y 448.198,Z 794.651,A -85,B 0,C 180,E1 -8744.065,E2 -8744.065} C_VEL
LIN {X 0,Y 448.865,Z 781.956,A -85,B 0,C 180,E1 -8744.855,E2 -8744.855} C_VEL
LIN {X 0,Y 449.34,Z 768.882,A -85,B 0,C 180,E1 -8745.448,E2 -8745.448} C_VEL
LIN {X 0,Y 449.855,Z 755.012,A -85,B 0,C 180,E1 -8745.866,E2 -8745.866} C_VEL
LIN {X 0,Y 450.662,Z 668.692,A -85,B 0,C 180,E1 -8747.344,E2 -8747.344} C_VEL
LIN {X 0,Y 447.411,Z 645.67,A -85,B 0,C 180,E1 -8747.908,E2 -8747.908} C_VEL
LIN {X 0,Y 448.371,Z 626.91,A -85,B 0,C 180,E1 -8751.131,E2 -8751.131} C_VEL
LIN {X 0,Y 449.325,Z 609.129,A -85,B 0,C 180,E1 -8754.24,E2 -8754.24} C_VEL
LIN {X 0,Y 449.502,Z 605.052,A -85,B 0,C 180,E1 -8754.969,E2 -8754.969} C_VEL
LIN {X 0,Y 447.169,Z 592.717,A -85,B 0,C 180,E1 -8757.367,E2 -8757.367} C_VEL
LIN {X 0,Y 446.498,Z 589.869,A -85,B 0,C 180,E1 -8757.963,E2 -8757.963} C_VEL
LIN {X 0,Y 446.414,Z 589.88,A -85,B 0,C 180,E1 -8761.299,E2 -8761.299} C_VEL
LIN {X 0,Y 446.428,Z 589.879,A -85,B 0,C 180,E1 -8764.522,E2 -8764.522} C_VEL
LIN {X 0,Y 446.434,Z 589.876,A -85,B 0,C 180,E1 -8768.082,E2 -8768.082} C_VEL
LIN {X 0,Y 446.439,Z 589.877,A -85,B 0,C 180,E1 -8770.919,E2 -8770.919} C_VEL
LIN {X 0,Y 446.397,Z 589.88,A -85,B 0,C 180,E1 -8773.845,E2 -8773.845} C_VEL
LIN {X 0,Y 446.442,Z 589.877,A -85,B 0,C 180,E1 -8776.396,E2 -8776.396} C_VEL
LIN {X 0,Y 446.464,Z 589.87,A -85,B 0,C 180,E1 -8779.804,E2 -8779.804} C_VEL
LIN {X 0,Y 446.429,Z 589.876,A -85,B 0,C 180,E1 -8782.123,E2 -8782.123} C_VEL
LIN {X 0,Y 446.424,Z 589.872,A -85,B 0,C 180,E1 -8785.476,E2 -8785.476} C_VEL
LIN {X 0,Y 446.424,Z 589.875,A -85,B 0,C 180,E1 -8788.7,E2 -8788.7} C_VEL
LIN {X 0,Y 446.477,Z 589.864,A -85,B 0,C 180,E1 -8791.821,E2 -8791.821} C_VEL
LIN {X 0,Y 446.451,Z 589.872,A -85,B 0,C 180,E1 -8794.847,E2 -8794.847} C_VEL
LIN {X 0,Y 446.44,Z 589.876,A -85,B 0,C 180,E1 -8798.244,E2 -8798.244} C_VEL
LIN {X 0,Y 446.45,Z 589.871,A -85,B 0,C 180,E1 -8801.649,E2 -8801.649} C_VEL
LIN {X 0,Y 446.499,Z 589.867,A -85,B 0,C 180,E1 -8804.479,E2 -8804.479} C_VEL
LIN {X 0,Y 446.531,Z 589.863,A -85,B 0,C 180,E1 -8808.193,E2 -8808.193} C_VEL
LIN {X 0,Y 446.592,Z 589.855,A -85,B 0,C 180,E1 -8811.858,E2 -8811.858} C_VEL
LIN {X 0,Y 446.638,Z 589.85,A -85,B 0,C 180,E1 -8814.582,E2 -8814.582} C_VEL
LIN {X 0,Y 446.702,Z 589.839,A -85,B 0,C 180,E1 -8817.295,E2 -8817.295} C_VEL
LIN {X 0,Y 446.786,Z 589.833,A -85,B 0,C 180,E1 -8820,E2 -8820} C_VEL
LIN {X 0,Y 446.702,Z 589.843,A -85,B 0,C 180,E1 -8822.705,E2 -8822.705} C_VEL
LIN {X 0,Y 446.644,Z 589.853,A -85,B 0,C 180,E1 -8826.324,E2 -8826.324} C_VEL
LIN {X 0,Y 446.531,Z 589.863,A -85,B 0,C 180,E1 -8829.055,E2 -8829.055} C_VEL
LIN {X 0,Y 446.522,Z 589.869,A -85,B 0,C 180,E1 -8832.73,E2 -8832.73} C_VEL
LIN {X 0,Y 446.517,Z 590.053,A -85,B 0,C 180,E1 -8834.702,E2 -8834.702} C_VEL
LIN {X 0,Y 447.685,Z 596.563,A -85,B 0,C 180,E1 -8836.414,E2 -8836.414} C_VEL
LIN {X 0,Y 447.799,Z 599.712,A -85,B 0,C 180,E1 -8837.205,E2 -8837.205} C_VEL
LIN {X 0,Y 451.175,Z 614.983,A -85,B 0,C 180,E1 -8837.634,E2 -8837.634} C_VEL
LIN {X 0,Y 450.078,Z 705.903,A -85,B 0,C 180,E1 -8839.201,E2 -8839.201} C_VEL
LIN {X 0,Y 449.742,Z 718.953,A -85,B 0,C 180,E1 -8839.602,E2 -8839.602} C_VEL
LIN {X 0,Y 449.312,Z 732.106,A -85,B 0,C 180,E1 -8840.203,E2 -8840.203} C_VEL
LIN {X 0,Y 448.824,Z 744.387,A -85,B 0,C 180,E1 -8840.977,E2 -8840.977} C_VEL
LIN {X 0,Y 448.294,Z 755.322,A -85,B 0,C 180,E1 -8841.86,E2 -8841.86} C_VEL
LIN {X 0,Y 447.706,Z 765.444,A -85,B 0,C 180,E1 -8842.875,E2 -8842.875} C_VEL
LIN {X 0,Y 447.121,Z 775.365,A -85,B 0,C 180,E1 -8844.122,E2 -8844.122} C_VEL
LIN {X 0,Y 446.624,Z 783.545,A -85,B 0,C 180,E1 -8845.391,E2 -8845.391} C_VEL
LIN {X 0,Y 446.284,Z 790.213,A -85,B 0,C 180,E1 -8846.667,E2 -8846.667} C_VEL
LIN {X 0,Y 445.934,Z 796.612,A -85,B 0,C 180,E1 -8848.216,E2 -8848.216} C_VEL
LIN {X 0,Y 445.681,Z 801.703,A -85,B 0,C 180,E1 -8849.856,E2 -8849.856} C_VEL
LIN {X 0,Y 445.524,Z 805.053,A -85,B 0,C 180,E1 -8851.37,E2 -8851.37} C_VEL
LIN {X 0,Y 445.444,Z 806.666,A -85,B 0,C 180,E1 -8852.441,E2 -8852.441} C_VEL
LIN {X 0,Y 445.344,Z 807.754,A -85,B 0,C 180,E1 -8853.527,E2 -8853.527} C_VEL
LIN {X 0,Y 445.321,Z 808.255,A -85,B 0,C 180,E1 -8854.852,E2 -8854.852} C_VEL
LIN {X 0,Y 445.33,Z 807.78,A -85,B 0,C 180,E1 -8856.405,E2 -8856.405} C_VEL
LIN {X 0,Y 445.399,Z 806.082,A -85,B 0,C 180,E1 -8857.98,E2 -8857.98} C_VEL
LIN {X 0,Y 445.61,Z 802.521,A -85,B 0,C 180,E1 -8859.798,E2 -8859.798} C_VEL
LIN {X 0,Y 445.817,Z 797.699,A -85,B 0,C 180,E1 -8861.46,E2 -8861.46} C_VEL
LIN {X 0,Y 446.052,Z 792.162,A -85,B 0,C 180,E1 -8862.885,E2 -8862.885} C_VEL
LIN {X 0,Y 446.486,Z 784.733,A -85,B 0,C 180,E1 -8864.386,E2 -8864.386} C_VEL
LIN {X 0,Y 446.916,Z 776.691,A -85,B 0,C 180,E1 -8865.685,E2 -8865.685} C_VEL
LIN {X 0,Y 447.483,Z 767.226,A -85,B 0,C 180,E1 -8866.912,E2 -8866.912} C_VEL
LIN {X 0,Y 448.061,Z 756.919,A -85,B 0,C 180,E1 -8867.995,E2 -8867.995} C_VEL
LIN {X 0,Y 448.585,Z 746.163,A -85,B 0,C 180,E1 -8868.903,E2 -8868.903} C_VEL
LIN {X 0,Y 449.12,Z 734.339,A -85,B 0,C 180,E1 -8869.682,E2 -8869.682} C_VEL
LIN {X 0,Y 449.541,Z 722.355,A -85,B 0,C 180,E1 -8870.282,E2 -8870.282} C_VEL
LIN {X 0,Y 449.829,Z 709.847,A -85,B 0,C 180,E1 -8870.73,E2 -8870.73} C_VEL
LIN {X 0,Y 450.074,Z 694.864,A -85,B 0,C 180,E1 -8871.044,E2 -8871.044} C_VEL
LIN {X 0,Y 450.888,Z 621.632,A -85,B 0,C 180,E1 -8872.271,E2 -8872.271} C_VEL
LIN {X 0,Y 450.102,Z 617.867,A -85,B 0,C 180,E1 -8872.366,E2 -8872.366} C_VEL
LIN {X 0,Y 446.83,Z 612.327,A -85,B 0,C 180,E1 -8872.591,E2 -8872.591} C_VEL
LIN {X 0,Y 443.088,Z 606.889,A -85,B 0,C 180,E1 -8872.836,E2 -8872.836} C_VEL
LIN {X 0,Y 441.612,Z 603.225,A -85,B 0,C 180,E1 -8872.96,E2 -8872.96} C_VEL
LIN {X 0,Y 440.611,Z 598.634,A -85,B 0,C 180,E1 -8873.096,E2 -8873.096} C_VEL
LIN {X 0,Y 439.798,Z 592.677,A -85,B 0,C 180,E1 -8874.586,E2 -8874.586} C_VEL
LIN {X 0,Y 439.439,Z 590.748,A -85,B 0,C 180,E1 -8875.129,E2 -8875.129} C_VEL
LIN {X 0,Y 439.369,Z 590.757,A -85,B 0,C 180,E1 -8878.141,E2 -8878.141} C_VEL
LIN {X 0,Y 439.429,Z 590.746,A -85,B 0,C 180,E1 -8881.599,E2 -8881.599} C_VEL
LIN {X 0,Y 439.403,Z 590.75,A -85,B 0,C 180,E1 -8884.416,E2 -8884.416} C_VEL
LIN {X 0,Y 439.363,Z 590.752,A -85,B 0,C 180,E1 -8887.426,E2 -8887.426} C_VEL
LIN {X 0,Y 439.44,Z 590.744,A -85,B 0,C 180,E1 -8890.664,E2 -8890.664} C_VEL
LIN {X 0,Y 439.461,Z 590.747,A -85,B 0,C 180,E1 -8894.226,E2 -8894.226} C_VEL
LIN {X 0,Y 439.507,Z 590.737,A -85,B 0,C 180,E1 -8898.003,E2 -8898.003} C_VEL
LIN {X 0,Y 439.548,Z 590.729,A -85,B 0,C 180,E1 -8901.727,E2 -8901.727} C_VEL
LIN {X 0,Y 439.622,Z 590.727,A -85,B 0,C 180,E1 -8904.497,E2 -8904.497} C_VEL
LIN {X 0,Y 439.637,Z 590.721,A -85,B 0,C 180,E1 -8908.169,E2 -8908.169} C_VEL
LIN {X 0,Y 439.764,Z 590.703,A -85,B 0,C 180,E1 -8910.001,E2 -8910.001} C_VEL
LIN {X 0,Y 439.658,Z 590.721,A -85,B 0,C 180,E1 -8912.75,E2 -8912.75} C_VEL
LIN {X 0,Y 439.621,Z 590.724,A -85,B 0,C 180,E1 -8916.426,E2 -8916.426} C_VEL
LIN {X 0,Y 439.503,Z 590.736,A -85,B 0,C 180,E1 -8919.202,E2 -8919.202} C_VEL
LIN {X 0,Y 439.468,Z 590.744,A -85,B 0,C 180,E1 -8922.938,E2 -8922.938} C_VEL
LIN {X 0,Y 439.45,Z 590.742,A -85,B 0,C 180,E1 -8926.35,E2 -8926.35} C_VEL
LIN {X 0,Y 439.406,Z 590.746,A -85,B 0,C 180,E1 -8929.627,E2 -8929.627} C_VEL
LIN {X 0,Y 439.368,Z 590.754,A -85,B 0,C 180,E1 -8932.576,E2 -8932.576} C_VEL
LIN {X 0,Y 439.409,Z 590.747,A -85,B 0,C 180,E1 -8935.586,E2 -8935.586} C_VEL
LIN {X 0,Y 439.421,Z 590.747,A -85,B 0,C 180,E1 -8938.674,E2 -8938.674} C_VEL
LIN {X 0,Y 439.374,Z 590.75,A -85,B 0,C 180,E1 -8942.031,E2 -8942.031} C_VEL
LIN {X 0,Y 439.399,Z 590.753,A -85,B 0,C 180,E1 -8945.341,E2 -8945.341} C_VEL
LIN {X 0,Y 439.387,Z 590.749,A -85,B 0,C 180,E1 -8948.595,E2 -8948.595} C_VEL
LIN {X 0,Y 439.392,Z 590.755,A -85,B 0,C 180,E1 -8951.257,E2 -8951.257} C_VEL
LIN {X 0,Y 439.404,Z 590.747,A -85,B 0,C 180,E1 -8954.73,E2 -8954.73} C_VEL
LIN {X 0,Y 439.4,Z 590.75,A -85,B 0,C 180,E1 -8957.796,E2 -8957.796} C_VEL
LIN {X 0,Y 439.399,Z 590.747,A -85,B 0,C 180,E1 -8960.224,E2 -8960.224} C_VEL
LIN {X 0,Y 439.378,Z 590.755,A -85,B 0,C 180,E1 -8963.713,E2 -8963.713} C_VEL
LIN {X 0,Y 439.377,Z 590.751,A -85,B 0,C 180,E1 -8967.054,E2 -8967.054} C_VEL
LIN {X 0,Y 439.387,Z 590.749,A -85,B 0,C 180,E1 -8970.275,E2 -8970.275} C_VEL
LIN {X 0,Y 439.433,Z 590.747,A -85,B 0,C 180,E1 -8973.397,E2 -8973.397} C_VEL
LIN {X 0,Y 439.389,Z 590.749,A -85,B 0,C 180,E1 -8976.43,E2 -8976.43} C_VEL
LIN {X 0,Y 439.393,Z 590.75,A -85,B 0,C 180,E1 -8979.397,E2 -8979.397} C_VEL
LIN {X 0,Y 439.431,Z 590.745,A -85,B 0,C 180,E1 -8982.31,E2 -8982.31} C_VEL
LIN {X 0,Y 439.453,Z 590.74,A -85,B 0,C 180,E1 -8985.174,E2 -8985.174} C_VEL
LIN {X 0,Y 439.489,Z 590.744,A -85,B 0,C 180,E1 -8988.002,E2 -8988.002} C_VEL
LIN {X 0,Y 439.553,Z 590.731,A -85,B 0,C 180,E1 -8991.726,E2 -8991.726} C_VEL
LIN {X 0,Y 439.624,Z 590.722,A -85,B 0,C 180,E1 -8994.496,E2 -8994.496} C_VEL
LIN {X 0,Y 439.639,Z 590.725,A -85,B 0,C 180,E1 -8998.168,E2 -8998.168} C_VEL
LIN {X 0,Y 439.768,Z 590.706,A -85,B 0,C 180,E1 -9000,E2 -9000} C_VEL
LIN {X 0,Y 439.646,Z 590.718,A -85,B 0,C 180,E1 -9002.749,E2 -9002.749} C_VEL
LIN {X 0,Y 439.623,Z 590.725,A -85,B 0,C 180,E1 -9006.425,E2 -9006.425} C_VEL
LIN {X 0,Y 439.504,Z 590.734,A -85,B 0,C 180,E1 -9009.202,E2 -9009.202} C_VEL
LIN {X 0,Y 439.471,Z 590.74,A -85,B 0,C 180,E1 -9012.938,E2 -9012.938} C_VEL
LIN {X 0,Y 439.452,Z 590.746,A -85,B 0,C 180,E1 -9016.348,E2 -9016.348} C_VEL
LIN {X 0,Y 439.408,Z 590.746,A -85,B 0,C 180,E1 -9019.626,E2 -9019.626} C_VEL
LIN {X 0,Y 439.371,Z 590.758,A -85,B 0,C 180,E1 -9022.575,E2 -9022.575} C_VEL
LIN {X 0,Y 439.406,Z 590.746,A -85,B 0,C 180,E1 -9025.585,E2 -9025.585} C_VEL
LIN {X 0,Y 439.423,Z 590.752,A -85,B 0,C 180,E1 -9028.673,E2 -9028.673} C_VEL
LIN {X 0,Y 439.376,Z 590.75,A -85,B 0,C 180,E1 -9032.03,E2 -9032.03} C_VEL
LIN {X 0,Y 439.4,Z 590.749,A -85,B 0,C 180,E1 -9035.34,E2 -9035.34} C_VEL
LIN {X 0,Y 439.383,Z 590.753,A -85,B 0,C 180,E1 -9038.595,E2 -9038.595} C_VEL
LIN {X 0,Y 439.394,Z 590.751,A -85,B 0,C 180,E1 -9041.256,E2 -9041.256} C_VEL
LIN {X 0,Y 439.407,Z 590.75,A -85,B 0,C 180,E1 -9044.729,E2 -9044.729} C_VEL
LIN {X 0,Y 439.401,Z 590.747,A -85,B 0,C 180,E1 -9047.795,E2 -9047.795} C_VEL
LIN {X 0,Y 439.431,Z 590.743,A -85,B 0,C 180,E1 -9050.227,E2 -9050.227} C_VEL
LIN {X 0,Y 439.379,Z 590.751,A -85,B 0,C 180,E1 -9053.712,E2 -9053.712} C_VEL
LIN {X 0,Y 439.378,Z 590.756,A -85,B 0,C 180,E1 -9057.054,E2 -9057.054} C_VEL
LIN {X 0,Y 439.387,Z 590.752,A -85,B 0,C 180,E1 -9060.274,E2 -9060.274} C_VEL
LIN {X 0,Y 439.478,Z 590.878,A -85,B 0,C 180,E1 -9061.793,E2 -9061.793} C_VEL
LIN {X 0,Y 442.191,Z 603.811,A -85,B 0,C 180,E1 -9064.335,E2 -9064.335} C_VEL
LIN {X 0,Y 442.654,Z 608.393,A -85,B 0,C 180,E1 -9065.192,E2 -9065.192} C_VEL
LIN {X 0,Y 441.595,Z 625.853,A -85,B 0,C 180,E1 -9068.282,E2 -9068.282} C_VEL
LIN {X 0,Y 440.691,Z 643.706,A -85,B 0,C 180,E1 -9071.399,E2 -9071.399} C_VEL
LIN {X 0,Y 440.539,Z 646.673,A -85,B 0,C 180,E1 -9071.914,E2 -9071.914} C_VEL
LIN {X 0,Y 443.881,Z 670.923,A -85,B 0,C 180,E1 -9072.475,E2 -9072.475} C_VEL
LIN {X 0,Y 442.947,Z 755.533,A -85,B 0,C 180,E1 -9073.937,E2 -9073.937} C_VEL
LIN {X 0,Y 442.491,Z 768.602,A -85,B 0,C 180,E1 -9074.334,E2 -9074.334} C_VEL
LIN {X 0,Y 441.985,Z 781.286,A -85,B 0,C 180,E1 -9074.907,E2 -9074.907} C_VEL
LIN {X 0,Y 441.366,Z 792.606,A -85,B 0,C 180,E1 -9075.592,E2 -9075.592} C_VEL
LIN {X 0,Y 440.736,Z 804.565,A -85,B 0,C 180,E1 -9076.534,E2 -9076.534} C_VEL
LIN {X 0,Y 440.104,Z 814.877,A -85,B 0,C 180,E1 -9077.549,E2 -9077.549} C_VEL
LIN {X 0,Y 439.631,Z 824.391,A -85,B 0,C 180,E1 -9078.706,E2 -9078.706} C_VEL
LIN {X 0,Y 439.088,Z 833.554,A -85,B 0,C 180,E1 -9080.091,E2 -9080.091} C_VEL
LIN {X 0,Y 438.788,Z 840.945,A -85,B 0,C 180,E1 -9081.479,E2 -9081.479} C_VEL
LIN {X 0,Y 438.54,Z 845.937,A -85,B 0,C 180,E1 -9082.633,E2 -9082.633} C_VEL
LIN {X 0,Y 438.396,Z 850.615,A -85,B 0,C 180,E1 -9083.965,E2 -9083.965} C_VEL
LIN {X 0,Y 438.357,Z 854.483,A -85,B 0,C 180,E1 -9085.401,E2 -9085.401} C_VEL
LIN {X 0,Y 438.329,Z 856.39,A -85,B 0,C 180,E1 -9086.322,E2 -9086.322} C_VEL
LIN {X 0,Y 438.392,Z 857.828,A -85,B 0,C 180,E1 -9087.242,E2 -9087.242} C_VEL
LIN {X 0,Y 438.366,Z 858.837,A -85,B 0,C 180,E1 -9088.162,E2 -9088.162} C_VEL
LIN {X 0,Y 438.366,Z 859.449,A -85,B 0,C 180,E1 -9089.08,E2 -9089.08} C_VEL
LIN {X 0,Y 438.337,Z 859.659,A -85,B 0,C 180,E1 -9089.999,E2 -9089.999} C_VEL
LIN {X 0,Y 438.366,Z 859.428,A -85,B 0,C 180,E1 -9090.918,E2 -9090.918} C_VEL
LIN {X 0,Y 438.367,Z 858.788,A -85,B 0,C 180,E1 -9091.836,E2 -9091.836} C_VEL
LIN {X 0,Y 438.397,Z 857.752,A -85,B 0,C 180,E1 -9092.756,E2 -9092.756} C_VEL
LIN {X 0,Y 438.328,Z 856.298,A -85,B 0,C 180,E1 -9093.676,E2 -9093.676} C_VEL
LIN {X 0,Y 438.422,Z 853.267,A -85,B 0,C 180,E1 -9095.057,E2 -9095.057} C_VEL
LIN {X 0,Y 438.448,Z 849.165,A -85,B 0,C 180,E1 -9096.441,E2 -9096.441} C_VEL
LIN {X 0,Y 438.67,Z 842.87,A -85,B 0,C 180,E1 -9098.057,E2 -9098.057} C_VEL
LIN {X 0,Y 438.97,Z 836.008,A -85,B 0,C 180,E1 -9099.444,E2 -9099.444} C_VEL
LIN {X 0,Y 439.388,Z 827.5,A -85,B 0,C 180,E1 -9100.832,E2 -9100.832} C_VEL
LIN {X 0,Y 439.957,Z 818.755,A -85,B 0,C 180,E1 -9101.984,E2 -9101.984} C_VEL
LIN {X 0,Y 440.477,Z 809.182,A -85,B 0,C 180,E1 -9103.023,E2 -9103.023} C_VEL
LIN {X 0,Y 441.082,Z 798.763,A -85,B 0,C 180,E1 -9103.944,E2 -9103.944} C_VEL
LIN {X 0,Y 441.638,Z 787.389,A -85,B 0,C 180,E1 -9104.75,E2 -9104.75} C_VEL
LIN {X 0,Y 442.184,Z 775.869,A -85,B 0,C 180,E1 -9105.379,E2 -9105.379} C_VEL
LIN {X 0,Y 442.765,Z 762.778,A -85,B 0,C 180,E1 -9105.89,E2 -9105.89} C_VEL
LIN {X 0,Y 443.127,Z 748.98,A -85,B 0,C 180,E1 -9106.231,E2 -9106.231} C_VEL
LIN {X 0,Y 443.89,Z 669.378,A -85,B 0,C 180,E1 -9107.613,E2 -9107.613} C_VEL
LIN {X 0,Y 440.487,Z 645.27,A -85,B 0,C 180,E1 -9108.21,E2 -9108.21} C_VEL
LIN {X 0,Y 441.408,Z 627.948,A -85,B 0,C 180,E1 -9111.235,E2 -9111.235} C_VEL
LIN {X 0,Y 442.499,Z 609.135,A -85,B 0,C 180,E1 -9114.592,E2 -9114.592} C_VEL
LIN {X 0,Y 442.36,Z 604.793,A -85,B 0,C 180,E1 -9115.4,E2 -9115.4} C_VEL
LIN {X 0,Y 439.885,Z 592.647,A -85,B 0,C 180,E1 -9117.837,E2 -9117.837} C_VEL
LIN {X 0,Y 439.452,Z 590.747,A -85,B 0,C 180,E1 -9118.258,E2 -9118.258} C_VEL
LIN {X 0,Y 439.371,Z 590.758,A -85,B 0,C 180,E1 -9121.859,E2 -9121.859} C_VEL
LIN {X 0,Y 439.398,Z 590.752,A -85,B 0,C 180,E1 -9125.155,E2 -9125.155} C_VEL
LIN {X 0,Y 439.394,Z 590.756,A -85,B 0,C 180,E1 -9128.592,E2 -9128.592} C_VEL
LIN {X 0,Y 439.394,Z 590.753,A -85,B 0,C 180,E1 -9131.257,E2 -9131.257} C_VEL
LIN {X 0,Y 439.398,Z 590.754,A -85,B 0,C 180,E1 -9134.728,E2 -9134.728} C_VEL
LIN {X 0,Y 439.407,Z 590.75,A -85,B 0,C 180,E1 -9137.797,E2 -9137.797} C_VEL
LIN {X 0,Y 439.447,Z 590.748,A -85,B 0,C 180,E1 -9140.229,E2 -9140.229} C_VEL
LIN {X 0,Y 439.371,Z 590.75,A -85,B 0,C 180,E1 -9143.712,E2 -9143.712} C_VEL
LIN {X 0,Y 439.369,Z 590.753,A -85,B 0,C 180,E1 -9147.053,E2 -9147.053} C_VEL
LIN {X 0,Y 439.39,Z 590.753,A -85,B 0,C 180,E1 -9150.275,E2 -9150.275} C_VEL
LIN {X 0,Y 439.426,Z 590.743,A -85,B 0,C 180,E1 -9153.588,E2 -9153.588} C_VEL
LIN {X 0,Y 439.38,Z 590.753,A -85,B 0,C 180,E1 -9156.429,E2 -9156.429} C_VEL
LIN {X 0,Y 439.381,Z 590.748,A -85,B 0,C 180,E1 -9159.397,E2 -9159.397} C_VEL
LIN {X 0,Y 439.424,Z 590.748,A -85,B 0,C 180,E1 -9162.309,E2 -9162.309} C_VEL
LIN {X 0,Y 439.439,Z 590.742,A -85,B 0,C 180,E1 -9165.174,E2 -9165.174} C_VEL
LIN {X 0,Y 439.499,Z 590.738,A -85,B 0,C 180,E1 -9168.002,E2 -9168.002} C_VEL
LIN {X 0,Y 439.539,Z 590.733,A -85,B 0,C 180,E1 -9171.726,E2 -9171.726} C_VEL
LIN {X 0,Y 439.613,Z 590.725,A -85,B 0,C 180,E1 -9174.496,E2 -9174.496} C_VEL
LIN {X 0,Y 439.628,Z 590.726,A -85,B 0,C 180,E1 -9178.168,E2 -9178.168} C_VEL
LIN {X 0,Y 439.756,Z 590.709,A -85,B 0,C 180,E1 -9180,E2 -9180} C_VEL
LIN {X 0,Y 439.649,Z 590.721,A -85,B 0,C 180,E1 -9182.749,E2 -9182.749} C_VEL
LIN {X 0,Y 439.614,Z 590.729,A -85,B 0,C 180,E1 -9186.425,E2 -9186.425} C_VEL
LIN {X 0,Y 439.493,Z 590.739,A -85,B 0,C 180,E1 -9189.202,E2 -9189.202} C_VEL
LIN {X 0,Y 439.487,Z 590.745,A -85,B 0,C 180,E1 -9192.722,E2 -9192.722} C_VEL
LIN {X 0,Y 439.446,Z 590.803,A -85,B 0,C 180,E1 -9194.412,E2 -9194.412} C_VEL
LIN {X 0,Y 440.698,Z 597.508,A -85,B 0,C 180,E1 -9196.205,E2 -9196.205} C_VEL
LIN {X 0,Y 440.919,Z 600.413,A -85,B 0,C 180,E1 -9196.907,E2 -9196.907} C_VEL
LIN {X 0,Y 444.443,Z 615.807,A -85,B 0,C 180,E1 -9197.352,E2 -9197.352} C_VEL
LIN {X 0,Y 443.275,Z 706.002,A -85,B 0,C 180,E1 -9198.937,E2 -9198.937} C_VEL
LIN {X 0,Y 442.926,Z 719.126,A -85,B 0,C 180,E1 -9199.343,E2 -9199.343} C_VEL
LIN {X 0,Y 442.489,Z 732.285,A -85,B 0,C 180,E1 -9199.951,E2 -9199.951} C_VEL
LIN {X 0,Y 442.001,Z 744.357,A -85,B 0,C 180,E1 -9200.719,E2 -9200.719} C_VEL
LIN {X 0,Y 441.434,Z 755.237,A -85,B 0,C 180,E1 -9201.603,E2 -9201.603} C_VEL
LIN {X 0,Y 440.823,Z 765.342,A -85,B 0,C 180,E1 -9202.62,E2 -9202.62} C_VEL
LIN {X 0,Y 440.216,Z 774.597,A -85,B 0,C 180,E1 -9203.773,E2 -9203.773} C_VEL
LIN {X 0,Y 439.701,Z 782.961,A -85,B 0,C 180,E1 -9205.06,E2 -9205.06} C_VEL
LIN {X 0,Y 439.311,Z 789.938,A -85,B 0,C 180,E1 -9206.382,E2 -9206.382} C_VEL
LIN {X 0,Y 438.948,Z 796.566,A -85,B 0,C 180,E1 -9207.966,E2 -9207.966} C_VEL
LIN {X 0,Y 438.689,Z 800.744,A -85,B 0,C 180,E1 -9209.25,E2 -9209.25} C_VEL
LIN {X 0,Y 438.495,Z 804.622,A -85,B 0,C 180,E1 -9210.856,E2 -9210.856} C_VEL
LIN {X 0,Y 438.385,Z 806.493,A -85,B 0,C 180,E1 -9211.941,E2 -9211.941} C_VEL
LIN {X 0,Y 438.271,Z 808.182,A -85,B 0,C 180,E1 -9213.505,E2 -9213.505} C_VEL
LIN {X 0,Y 438.253,Z 808.651,A -85,B 0,C 180,E1 -9215.262,E2 -9215.262} C_VEL
LIN {X 0,Y 438.26,Z 807.966,A -85,B 0,C 180,E1 -9216.699,E2 -9216.699} C_VEL
LIN {X 0,Y 438.329,Z 806.157,A -85,B 0,C 180,E1 -9218.221,E2 -9218.221} C_VEL
LIN {X 0,Y 438.545,Z 802.903,A -85,B 0,C 180,E1 -9219.869,E2 -9219.869} C_VEL
LIN {X 0,Y 438.788,Z 797.65,A -85,B 0,C 180,E1 -9221.674,E2 -9221.674} C_VEL
LIN {X 0,Y 439.072,Z 791.487,A -85,B 0,C 180,E1 -9223.237,E2 -9223.237} C_VEL
LIN {X 0,Y 439.527,Z 784.048,A -85,B 0,C 180,E1 -9224.713,E2 -9224.713} C_VEL
LIN {X 0,Y 440.01,Z 776.256,A -85,B 0,C 180,E1 -9225.952,E2 -9225.952} C_VEL
LIN {X 0,Y 440.576,Z 766.571,A -85,B 0,C 180,E1 -9227.205,E2 -9227.205} C_VEL
LIN {X 0,Y 441.12,Z 757.237,A -85,B 0,C 180,E1 -9228.187,E2 -9228.187} C_VEL
LIN {X 0,Y 441.673,Z 746.669,A -85,B 0,C 180,E1 -9229.093,E2 -9229.093} C_VEL
LIN {X 0,Y 442.242,Z 734.797,A -85,B 0,C 180,E1 -9229.888,E2 -9229.888} C_VEL
LIN {X 0,Y 442.676,Z 722.692,A -85,B 0,C 180,E1 -9230.504,E2 -9230.504} C_VEL
LIN {X 0,Y 442.988,Z 709.828,A -85,B 0,C 180,E1 -9230.969,E2 -9230.969} C_VEL
LIN {X 0,Y 443.227,Z 693.439,A -85,B 0,C 180,E1 -9231.307,E2 -9231.307} C_VEL
LIN {X 0,Y 444.148,Z 615.046,A -85,B 0,C 180,E1 -9232.648,E2 -9232.648} C_VEL
LIN {X 0,Y 441.612,Z 603.225,A -85,B 0,C 180,E1 -9232.96,E2 -9232.96} C_VEL
LIN {X 0,Y 440.457,Z 600.536,A -85,B 0,C 180,E1 -9233.119,E2 -9233.119} C_VEL
LIN {X 0,Y 438.105,Z 597.883,A -85,B 0,C 180,E1 -9233.498,E2 -9233.498} C_VEL
LIN {X 0,Y 435.27,Z 595.848,A -85,B 0,C 180,E1 -9234.063,E2 -9234.063} C_VEL
LIN {X 0,Y 433.067,Z 593.688,A -85,B 0,C 180,E1 -9234.714,E2 -9234.714} C_VEL
LIN {X 0,Y 432.542,Z 592.416,A -85,B 0,C 180,E1 -9235.052,E2 -9235.052} C_VEL
LIN {X 0,Y 432.39,Z 591.627,A -85,B 0,C 180,E1 -9235.329,E2 -9235.329} C_VEL
LIN {X 0,Y 432.317,Z 591.63,A -85,B 0,C 180,E1 -9238.655,E2 -9238.655} C_VEL
LIN {X 0,Y 432.379,Z 591.627,A -85,B 0,C 180,E1 -9241.878,E2 -9241.878} C_VEL
LIN {X 0,Y 432.349,Z 591.625,A -85,B 0,C 180,E1 -9245,E2 -9245} C_VEL
LIN {X 0,Y 432.356,Z 591.631,A -85,B 0,C 180,E1 -9248.047,E2 -9248.047} C_VEL
LIN {X 0,Y 432.385,Z 591.621,A -85,B 0,C 180,E1 -9251.031,E2 -9251.031} C_VEL
LIN {X 0,Y 432.43,Z 591.619,A -85,B 0,C 180,E1 -9253.962,E2 -9253.962} C_VEL
LIN {X 0,Y 432.48,Z 591.61,A -85,B 0,C 180,E1 -9257.805,E2 -9257.805} C_VEL
LIN {X 0,Y 432.492,Z 591.607,A -85,B 0,C 180,E1 -9261.591,E2 -9261.591} C_VEL
LIN {X 0,Y 432.598,Z 591.602,A -85,B 0,C 180,E1 -9264.407,E2 -9264.407} C_VEL
LIN {X 0,Y 432.607,Z 591.596,A -85,B 0,C 180,E1 -9268.139,E2 -9268.139} C_VEL
LIN {X 0,Y 432.733,Z 591.579,A -85,B 0,C 180,E1 -9270.001,E2 -9270.001} C_VEL
LIN {X 0,Y 432.607,Z 591.598,A -85,B 0,C 180,E1 -9272.795,E2 -9272.795} C_VEL
LIN {X 0,Y 432.575,Z 591.603,A -85,B 0,C 180,E1 -9276.531,E2 -9276.531} C_VEL
LIN {X 0,Y 432.446,Z 591.614,A -85,B 0,C 180,E1 -9279.354,E2 -9279.354} C_VEL
LIN {X 0,Y 432.434,Z 591.622,A -85,B 0,C 180,E1 -9282.804,E2 -9282.804} C_VEL
LIN {X 0,Y 432.415,Z 591.62,A -85,B 0,C 180,E1 -9286.48,E2 -9286.48} C_VEL
LIN {X 0,Y 432.342,Z 591.626,A -85,B 0,C 180,E1 -9289.961,E2 -9289.961} C_VEL
LIN {X 0,Y 432.322,Z 591.637,A -85,B 0,C 180,E1 -9292.965,E2 -9292.965} C_VEL
LIN {X 0,Y 432.368,Z 591.622,A -85,B 0,C 180,E1 -9296.033,E2 -9296.033} C_VEL
LIN {X 0,Y 432.347,Z 591.632,A -85,B 0,C 180,E1 -9299.188,E2 -9299.188} C_VEL
LIN {X 0,Y 432.327,Z 591.628,A -85,B 0,C 180,E1 -9302.444,E2 -9302.444} C_VEL
LIN {X 0,Y 432.348,Z 591.628,A -85,B 0,C 180,E1 -9305.633,E2 -9305.633} C_VEL
LIN {X 0,Y 432.354,Z 591.631,A -85,B 0,C 180,E1 -9309.343,E2 -9309.343} C_VEL
LIN {X 0,Y 432.337,Z 591.629,A -85,B 0,C 180,E1 -9311.798,E2 -9311.798} C_VEL
LIN {X 0,Y 432.337,Z 591.626,A -85,B 0,C 180,E1 -9314.348,E2 -9314.348} C_VEL
LIN {X 0,Y 432.324,Z 591.631,A -85,B 0,C 180,E1 -9317.016,E2 -9317.016} C_VEL
LIN {X 0,Y 432.338,Z 591.63,A -85,B 0,C 180,E1 -9319.821,E2 -9319.821} C_VEL
LIN {X 0,Y 432.31,Z 591.632,A -85,B 0,C 180,E1 -9323.022,E2 -9323.022} C_VEL
LIN {X 0,Y 432.364,Z 591.626,A -85,B 0,C 180,E1 -9325.997,E2 -9325.997} C_VEL
LIN {X 0,Y 432.352,Z 591.631,A -85,B 0,C 180,E1 -9329.49,E2 -9329.49} C_VEL
LIN {X 0,Y 432.395,Z 591.62,A -85,B 0,C 180,E1 -9332.929,E2 -9332.929} C_VEL
LIN {X 0,Y 432.373,Z 591.626,A -85,B 0,C 180,E1 -9336.024,E2 -9336.024} C_VEL
LIN {X 0,Y 432.355,Z 591.625,A -85,B 0,C 180,E1 -9339.046,E2 -9339.046} C_VEL
LIN {X 0,Y 432.379,Z 591.627,A -85,B 0,C 180,E1 -9342.011,E2 -9342.011} C_VEL
LIN {X 0,Y 432.4,Z 591.618,A -85,B 0,C 180,E1 -9344.927,E2 -9344.927} C_VEL
LIN {X 0,Y 432.464,Z 591.616,A -85,B 0,C 180,E1 -9347.804,E2 -9347.804} C_VEL
LIN {X 0,Y 432.497,Z 591.609,A -85,B 0,C 180,E1 -9351.591,E2 -9351.591} C_VEL
LIN {X 0,Y 432.6,Z 591.597,A -85,B 0,C 180,E1 -9354.406,E2 -9354.406} C_VEL
LIN {X 0,Y 432.609,Z 591.601,A -85,B 0,C 180,E1 -9358.138,E2 -9358.138} C_VEL
LIN {X 0,Y 432.738,Z 591.582,A -85,B 0,C 180,E1 -9360,E2 -9360} C_VEL
LIN {X 0,Y 432.597,Z 591.596,A -85,B 0,C 180,E1 -9362.794,E2 -9362.794} C_VEL
LIN {X 0,Y 432.578,Z 591.601,A -85,B 0,C 180,E1 -9366.53,E2 -9366.53} C_VEL
LIN {X 0,Y 432.447,Z 591.613,A -85,B 0,C 180,E1 -9369.353,E2 -9369.353} C_VEL
LIN {X 0,Y 432.437,Z 591.617,A -85,B 0,C 180,E1 -9372.803,E2 -9372.803} C_VEL
LIN {X 0,Y 432.418,Z 591.625,A -85,B 0,C 180,E1 -9376.478,E2 -9376.478} C_VEL
LIN {X 0,Y 432.344,Z 591.627,A -85,B 0,C 180,E1 -9379.96,E2 -9379.96} C_VEL
LIN {X 0,Y 432.325,Z 591.631,A -85,B 0,C 180,E1 -9382.964,E2 -9382.964} C_VEL
LIN {X 0,Y 432.368,Z 591.624,A -85,B 0,C 180,E1 -9386.032,E2 -9386.032} C_VEL
LIN {X 0,Y 432.349,Z 591.627,A -85,B 0,C 180,E1 -9389.187,E2 -9389.187} C_VEL
LIN {X 0,Y 432.329,Z 591.631,A -85,B 0,C 180,E1 -9392.443,E2 -9392.443} C_VEL
LIN {X 0,Y 432.35,Z 591.625,A -85,B 0,C 180,E1 -9395.632,E2 -9395.632} C_VEL
LIN {X 0,Y 432.346,Z 591.631,A -85,B 0,C 180,E1 -9398.714,E2 -9398.714} C_VEL
LIN {X 0,Y 432.339,Z 591.626,A -85,B 0,C 180,E1 -9401.797,E2 -9401.797} C_VEL
LIN {X 0,Y 432.339,Z 591.627,A -85,B 0,C 180,E1 -9404.347,E2 -9404.347} C_VEL
LIN {X 0,Y 432.326,Z 591.636,A -85,B 0,C 180,E1 -9407.015,E2 -9407.015} C_VEL
LIN {X 0,Y 432.338,Z 591.627,A -85,B 0,C 180,E1 -9409.82,E2 -9409.82} C_VEL
LIN {X 0,Y 432.312,Z 591.636,A -85,B 0,C 180,E1 -9413.022,E2 -9413.022} C_VEL
LIN {X 0,Y 432.365,Z 591.626,A -85,B 0,C 180,E1 -9415.996,E2 -9415.996} C_VEL
LIN {X 0,Y 432.352,Z 591.63,A -85,B 0,C 180,E1 -9419.489,E2 -9419.489} C_VEL
LIN {X 0,Y 432.393,Z 591.668,A -85,B 0,C 180,E1 -9421.53,E2 -9421.53} C_VEL
LIN {X 0,Y 435.143,Z 604.734,A -85,B 0,C 180,E1 -9424.145,E2 -9424.145} C_VEL
LIN {X 0,Y 435.696,Z 608.76,A -85,B 0,C 180,E1 -9424.919,E2 -9424.919} C_VEL
LIN {X 0,Y 434.89,Z 622.674,A -85,B 0,C 180,E1 -9427.429,E2 -9427.429} C_VEL
LIN {X 0,Y 433.879,Z 640.509,A -85,B 0,C 180,E1 -9430.605,E2 -9430.605} C_VEL
LIN {X 0,Y 433.599,Z 646.262,A -85,B 0,C 180,E1 -9431.623,E2 -9431.623} C_VEL
LIN {X 0,Y 437.053,Z 671.846,A -85,B 0,C 180,E1 -9432.234,E2 -9432.234} C_VEL
LIN {X 0,Y 436.075,Z 755.435,A -85,B 0,C 180,E1 -9433.707,E2 -9433.707} C_VEL
LIN {X 0,Y 435.583,Z 769.151,A -85,B 0,C 180,E1 -9434.139,E2 -9434.139} C_VEL
LIN {X 0,Y 435.047,Z 781.576,A -85,B 0,C 180,E1 -9434.72,E2 -9434.72} C_VEL
LIN {X 0,Y 434.361,Z 793.5,A -85,B 0,C 180,E1 -9435.475,E2 -9435.475} C_VEL
LIN {X 0,Y 433.77,Z 804.102,A -85,B 0,C 180,E1 -9436.331,E2 -9436.331} C_VEL
LIN {X 0,Y 433.158,Z 814.279,A -85,B 0,C 180,E1 -9437.347,E2 -9437.347} C_VEL
LIN {X 0,Y 432.604,Z 823.835,A -85,B 0,C 180,E1 -9438.52,E2 -9438.52} C_VEL
LIN {X 0,Y 432.038,Z 833.03,A -85,B 0,C 180,E1 -9439.928,E2 -9439.928} C_VEL
LIN {X 0,Y 431.718,Z 840.445,A -85,B 0,C 180,E1 -9441.338,E2 -9441.338} C_VEL
LIN {X 0,Y 431.467,Z 845.458,A -85,B 0,C 180,E1 -9442.512,E2 -9442.512} C_VEL
LIN {X 0,Y 431.297,Z 850.583,A -85,B 0,C 180,E1 -9444.005,E2 -9444.005} C_VEL
LIN {X 0,Y 431.288,Z 854.039,A -85,B 0,C 180,E1 -9445.326,E2 -9445.326} C_VEL
LIN {X 0,Y 431.234,Z 855.951,A -85,B 0,C 180,E1 -9446.261,E2 -9446.261} C_VEL
LIN {X 0,Y 431.318,Z 857.401,A -85,B 0,C 180,E1 -9447.197,E2 -9447.197} C_VEL
LIN {X 0,Y 431.285,Z 858.415,A -85,B 0,C 180,E1 -9448.131,E2 -9448.131} C_VEL
LIN {X 0,Y 431.276,Z 859.03,A -85,B 0,C 180,E1 -9449.065,E2 -9449.065} C_VEL
LIN {X 0,Y 431.277,Z 859.246,A -85,B 0,C 180,E1 -9449.999,E2 -9449.999} C_VEL
LIN {X 0,Y 431.276,Z 859.018,A -85,B 0,C 180,E1 -9450.933,E2 -9450.933} C_VEL
LIN {X 0,Y 431.287,Z 858.38,A -85,B 0,C 180,E1 -9451.867,E2 -9451.867} C_VEL
LIN {X 0,Y 431.323,Z 857.344,A -85,B 0,C 180,E1 -9452.801,E2 -9452.801} C_VEL
LIN {X 0,Y 431.232,Z 855.89,A -85,B 0,C 180,E1 -9453.737,E2 -9453.737} C_VEL
LIN {X 0,Y 431.328,Z 852.856,A -85,B 0,C 180,E1 -9455.14,E2 -9455.14} C_VEL
LIN {X 0,Y 431.376,Z 848.753,A -85,B 0,C 180,E1 -9456.547,E2 -9456.547} C_VEL
LIN {X 0,Y 431.603,Z 842.455,A -85,B 0,C 180,E1 -9458.19,E2 -9458.19} C_VEL
LIN {X 0,Y 431.912,Z 835.584,A -85,B 0,C 180,E1 -9459.6,E2 -9459.6} C_VEL
LIN {X 0,Y 432.387,Z 827.073,A -85,B 0,C 180,E1 -9461.009,E2 -9461.009} C_VEL
LIN {X 0,Y 432.961,Z 818.322,A -85,B 0,C 180,E1 -9462.181,E2 -9462.181} C_VEL
LIN {X 0,Y 433.556,Z 807.382,A -85,B 0,C 180,E1 -9463.372,E2 -9463.372} C_VEL
LIN {X 0,Y 434.226,Z 796.914,A -85,B 0,C 180,E1 -9464.288,E2 -9464.288} C_VEL
LIN {X 0,Y 434.867,Z 785.151,A -85,B 0,C 180,E1 -9465.105,E2 -9465.105} C_VEL
LIN {X 0,Y 435.395,Z 772.993,A -85,B 0,C 180,E1 -9465.745,E2 -9465.745} C_VEL
LIN {X 0,Y 436.021,Z 759.886,A -85,B 0,C 180,E1 -9466.232,E2 -9466.232} C_VEL
LIN {X 0,Y 436.349,Z 745.794,A -85,B 0,C 180,E1 -9466.551,E2 -9466.551} C_VEL
LIN {X 0,Y 437.138,Z 669.9,A -85,B 0,C 180,E1 -9467.894,E2 -9467.894} C_VEL
LIN {X 0,Y 433.554,Z 644.731,A -85,B 0,C 180,E1 -9468.545,E2 -9468.545} C_VEL
LIN {X 0,Y 434.598,Z 626.306,A -85,B 0,C 180,E1 -9471.834,E2 -9471.834} C_VEL
LIN {X 0,Y 435.678,Z 608.902,A -85,B 0,C 180,E1 -9475.001,E2 -9475.001} C_VEL
LIN {X 0,Y 434.88,Z 603.211,A -85,B 0,C 180,E1 -9476.127,E2 -9476.127} C_VEL
LIN {X 0,Y 432.881,Z 593.723,A -85,B 0,C 180,E1 -9478.087,E2 -9478.087} C_VEL
LIN {X 0,Y 432.393,Z 591.628,A -85,B 0,C 180,E1 -9478.539,E2 -9478.539} C_VEL
LIN {X 0,Y 432.319,Z 591.637,A -85,B 0,C 180,E1 -9481.345,E2 -9481.345} C_VEL
LIN {X 0,Y 432.338,Z 591.633,A -85,B 0,C 180,E1 -9484.676,E2 -9484.676} C_VEL
LIN {X 0,Y 432.349,Z 591.631,A -85,B 0,C 180,E1 -9488.147,E2 -9488.147} C_VEL
LIN {X 0,Y 432.362,Z 591.628,A -85,B 0,C 180,E1 -9491.606,E2 -9491.606} C_VEL
LIN {X 0,Y 432.373,Z 591.626,A -85,B 0,C 180,E1 -9495.657,E2 -9495.657} C_VEL
LIN {X 0,Y 432.368,Z 591.629,A -85,B 0,C 180,E1 -9498.391,E2 -9498.391} C_VEL
LIN {X 0,Y 432.348,Z 591.627,A -85,B 0,C 180,E1 -9501.851,E2 -9501.851} C_VEL
LIN {X 0,Y 432.335,Z 591.628,A -85,B 0,C 180,E1 -9505.322,E2 -9505.322} C_VEL
LIN {X 0,Y 432.326,Z 591.63,A -85,B 0,C 180,E1 -9508.654,E2 -9508.654} C_VEL
LIN {X 0,Y 432.377,Z 591.62,A -85,B 0,C 180,E1 -9511.876,E2 -9511.876} C_VEL
LIN {X 0,Y 432.344,Z 591.628,A -85,B 0,C 180,E1 -9514.998,E2 -9514.998} C_VEL
LIN {X 0,Y 432.35,Z 591.628,A -85,B 0,C 180,E1 -9518.045,E2 -9518.045} C_VEL
LIN {X 0,Y 432.379,Z 591.624,A -85,B 0,C 180,E1 -9521.029,E2 -9521.029} C_VEL
LIN {X 0,Y 432.422,Z 591.62,A -85,B 0,C 180,E1 -9523.961,E2 -9523.961} C_VEL
LIN {X 0,Y 432.472,Z 591.612,A -85,B 0,C 180,E1 -9527.804,E2 -9527.804} C_VEL
LIN {X 0,Y 432.484,Z 591.611,A -85,B 0,C 180,E1 -9531.59,E2 -9531.59} C_VEL
LIN {X 0,Y 432.59,Z 591.601,A -85,B 0,C 180,E1 -9534.406,E2 -9534.406} C_VEL
LIN {X 0,Y 432.597,Z 591.602,A -85,B 0,C 180,E1 -9538.138,E2 -9538.138} C_VEL
LIN {X 0,Y 432.726,Z 591.584,A -85,B 0,C 180,E1 -9540,E2 -9540} C_VEL
LIN {X 0,Y 432.598,Z 591.599,A -85,B 0,C 180,E1 -9542.793,E2 -9542.793} C_VEL
LIN {X 0,Y 432.568,Z 591.607,A -85,B 0,C 180,E1 -9546.53,E2 -9546.53} C_VEL
LIN {X 0,Y 432.437,Z 591.618,A -85,B 0,C 180,E1 -9549.353,E2 -9549.353} C_VEL
LIN {X 0,Y 432.431,Z 591.625,A -85,B 0,C 180,E1 -9552.809,E2 -9552.809} C_VEL
LIN {X 0,Y 432.434,Z 591.807,A -85,B 0,C 180,E1 -9554.17,E2 -9554.17} C_VEL
LIN {X 0,Y 433.728,Z 598.488,A -85,B 0,C 180,E1 -9555.99,E2 -9555.99} C_VEL
LIN {X 0,Y 433.918,Z 600.65,A -85,B 0,C 180,E1 -9556.556,E2 -9556.556} C_VEL
LIN {X 0,Y 437.336,Z 614.616,A -85,B 0,C 180,E1 -9557.004,E2 -9557.004} C_VEL
LIN {X 0,Y 437.723,Z 618.514,A -85,B 0,C 180,E1 -9557.096,E2 -9557.096} C_VEL
LIN {X 0,Y 436.479,Z 707.298,A -85,B 0,C 180,E1 -9558.693,E2 -9558.693} C_VEL
LIN {X 0,Y 436.123,Z 720.912,A -85,B 0,C 180,E1 -9559.137,E2 -9559.137} C_VEL
LIN {X 0,Y 435.648,Z 733.437,A -85,B 0,C 180,E1 -9559.741,E2 -9559.741} C_VEL
LIN {X 0,Y 435.085,Z 746.118,A -85,B 0,C 180,E1 -9560.578,E2 -9560.578} C_VEL
LIN {X 0,Y 434.529,Z 756.626,A -85,B 0,C 180,E1 -9561.465,E2 -9561.465} C_VEL
LIN {X 0,Y 433.816,Z 767.149,A -85,B 0,C 180,E1 -9562.572,E2 -9562.572} C_VEL
LIN {X 0,Y 433.231,Z 775.642,A -85,B 0,C 180,E1 -9563.672,E2 -9563.672} C_VEL
LIN {X 0,Y 432.68,Z 783.905,A -85,B 0,C 180,E1 -9564.981,E2 -9564.981} C_VEL
LIN {X 0,Y 432.289,Z 790.698,A -85,B 0,C 180,E1 -9566.307,E2 -9566.307} C_VEL
LIN {X 0,Y 431.937,Z 796.188,A -85,B 0,C 180,E1 -9567.627,E2 -9567.627} C_VEL
LIN {X 0,Y 431.629,Z 801.419,A -85,B 0,C 180,E1 -9569.24,E2 -9569.24} C_VEL
LIN {X 0,Y 431.427,Z 805.219,A -85,B 0,C 180,E1 -9570.873,E2 -9570.873} C_VEL
LIN {X 0,Y 431.246,Z 807.739,A -85,B 0,C 180,E1 -9572.534,E2 -9572.534} C_VEL
LIN {X 0,Y 431.162,Z 808.766,A -85,B 0,C 180,E1 -9573.769,E2 -9573.769} C_VEL
LIN {X 0,Y 431.156,Z 809.034,A -85,B 0,C 180,E1 -9575.413,E2 -9575.413} C_VEL
LIN {X 0,Y 431.192,Z 808.043,A -85,B 0,C 180,E1 -9577.09,E2 -9577.09} C_VEL
LIN {X 0,Y 431.279,Z 806.119,A -85,B 0,C 180,E1 -9578.54,E2 -9578.54} C_VEL
LIN {X 0,Y 431.496,Z 803.034,A -85,B 0,C 180,E1 -9580.049,E2 -9580.049} C_VEL
LIN {X 0,Y 431.685,Z 798.923,A -85,B 0,C 180,E1 -9581.507,E2 -9581.507} C_VEL
LIN {X 0,Y 431.988,Z 792.968,A -85,B 0,C 180,E1 -9583.102,E2 -9583.102} C_VEL
LIN {X 0,Y 432.476,Z 785.501,A -85,B 0,C 180,E1 -9584.655,E2 -9584.655} C_VEL
LIN {X 0,Y 433.02,Z 776.766,A -85,B 0,C 180,E1 -9586.092,E2 -9586.092} C_VEL
LIN {X 0,Y 433.651,Z 766.507,A -85,B 0,C 180,E1 -9587.435,E2 -9587.435} C_VEL
LIN {X 0,Y 434.234,Z 757.117,A -85,B 0,C 180,E1 -9588.428,E2 -9588.428} C_VEL
LIN {X 0,Y 434.781,Z 747.138,A -85,B 0,C 180,E1 -9589.291,E2 -9589.291} C_VEL
LIN {X 0,Y 435.324,Z 735.95,A -85,B 0,C 180,E1 -9590.061,E2 -9590.061} C_VEL
LIN {X 0,Y 435.813,Z 723.337,A -85,B 0,C 180,E1 -9590.719,E2 -9590.719} C_VEL
LIN {X 0,Y 436.138,Z 710.83,A -85,B 0,C 180,E1 -9591.184,E2 -9591.184} C_VEL
LIN {X 0,Y 436.374,Z 696.584,A -85,B 0,C 180,E1 -9591.5,E2 -9591.5} C_VEL
LIN {X 0,Y 437.219,Z 615.245,A -85,B 0,C 180,E1 -9592.922,E2 -9592.922} C_VEL
LIN {X 0,Y 433.652,Z 599.025,A -85,B 0,C 180,E1 -9593.375,E2 -9593.375} C_VEL
LIN {X 0,Y 432.542,Z 592.416,A -85,B 0,C 180,E1 -9595.052,E2 -9595.052} C_VEL
LIN {X 0,Y 432.115,Z 591.732,A -85,B 0,C 180,E1 -9595.406,E2 -9595.406} C_VEL
LIN {X 0,Y 429.739,Z 591.954,A -85,B 0,C 180,E1 -9596.527,E2 -9596.527} C_VEL
LIN {X 0,Y 426.233,Z 592.538,A -85,B 0,C 180,E1 -9598.077,E2 -9598.077} C_VEL
LIN {X 0,Y 425.333,Z 592.516,A -85,B 0,C 180,E1 -9598.887,E2 -9598.887} C_VEL
LIN {X 0,Y 425.281,Z 592.506,A -85,B 0,C 180,E1 -9599.16,E2 -9599.16} C_VEL
LIN {X 0,Y 425.346,Z 592.5,A -85,B 0,C 180,E1 -9602.443,E2 -9602.443} C_VEL
LIN {X 0,Y 425.349,Z 592.499,A -85,B 0,C 180,E1 -9605.603,E2 -9605.603} C_VEL
LIN {X 0,Y 425.292,Z 592.506,A -85,B 0,C 180,E1 -9608.683,E2 -9608.683} C_VEL
LIN {X 0,Y 425.332,Z 592.501,A -85,B 0,C 180,E1 -9611.704,E2 -9611.704} C_VEL
LIN {X 0,Y 425.348,Z 592.5,A -85,B 0,C 180,E1 -9614.672,E2 -9614.672} C_VEL
LIN {X 0,Y 425.43,Z 592.487,A -85,B 0,C 180,E1 -9617.6,E2 -9617.6} C_VEL
LIN {X 0,Y 425.443,Z 592.485,A -85,B 0,C 180,E1 -9621.451,E2 -9621.451} C_VEL
LIN {X 0,Y 425.555,Z 592.478,A -85,B 0,C 180,E1 -9624.314,E2 -9624.314} C_VEL
LIN {X 0,Y 425.577,Z 592.471,A -85,B 0,C 180,E1 -9628.108,E2 -9628.108} C_VEL
LIN {X 0,Y 425.703,Z 592.454,A -85,B 0,C 180,E1 -9630.001,E2 -9630.001} C_VEL
LIN {X 0,Y 425.559,Z 592.476,A -85,B 0,C 180,E1 -9632.841,E2 -9632.841} C_VEL
LIN {X 0,Y 425.533,Z 592.482,A -85,B 0,C 180,E1 -9636.64,E2 -9636.64} C_VEL
LIN {X 0,Y 425.404,Z 592.49,A -85,B 0,C 180,E1 -9639.51,E2 -9639.51} C_VEL
LIN {X 0,Y 425.396,Z 592.497,A -85,B 0,C 180,E1 -9642.905,E2 -9642.905} C_VEL
LIN {X 0,Y 425.364,Z 592.5,A -85,B 0,C 180,E1 -9646.606,E2 -9646.606} C_VEL
LIN {X 0,Y 425.332,Z 592.5,A -85,B 0,C 180,E1 -9649.637,E2 -9649.637} C_VEL
LIN {X 0,Y 425.31,Z 592.505,A -85,B 0,C 180,E1 -9653.366,E2 -9653.366} C_VEL
LIN {X 0,Y 425.351,Z 592.502,A -85,B 0,C 180,E1 -9656.845,E2 -9656.845} C_VEL
LIN {X 0,Y 425.295,Z 592.505,A -85,B 0,C 180,E1 -9659.72,E2 -9659.72} C_VEL
LIN {X 0,Y 425.286,Z 592.511,A -85,B 0,C 180,E1 -9663.049,E2 -9663.049} C_VEL
LIN {X 0,Y 425.286,Z 592.505,A -85,B 0,C 180,E1 -9665.929,E2 -9665.929} C_VEL
LIN {X 0,Y 425.301,Z 592.508,A -85,B 0,C 180,E1 -9669.044,E2 -9669.044} C_VEL
LIN {X 0,Y 425.279,Z 592.507,A -85,B 0,C 180,E1 -9672.654,E2 -9672.654} C_VEL
LIN {X 0,Y 425.265,Z 592.508,A -85,B 0,C 180,E1 -9676.045,E2 -9676.045} C_VEL
LIN {X 0,Y 425.278,Z 592.506,A -85,B 0,C 180,E1 -9678.622,E2 -9678.622} C_VEL
LIN {X 0,Y 425.301,Z 592.506,A -85,B 0,C 180,E1 -9681.102,E2 -9681.102} C_VEL
LIN {X 0,Y 425.304,Z 592.503,A -85,B 0,C 180,E1 -9684.665,E2 -9684.665} C_VEL
LIN {X 0,Y 425.269,Z 592.509,A -85,B 0,C 180,E1 -9688.074,E2 -9688.074} C_VEL
LIN {X 0,Y 425.336,Z 592.503,A -85,B 0,C 180,E1 -9691.368,E2 -9691.368} C_VEL
LIN {X 0,Y 425.358,Z 592.501,A -85,B 0,C 180,E1 -9693.506,E2 -9693.506} C_VEL
LIN {X 0,Y 425.29,Z 592.504,A -85,B 0,C 180,E1 -9696.634,E2 -9696.634} C_VEL
LIN {X 0,Y 425.3,Z 592.509,A -85,B 0,C 180,E1 -9699.695,E2 -9699.695} C_VEL
LIN {X 0,Y 425.345,Z 592.498,A -85,B 0,C 180,E1 -9702.698,E2 -9702.698} C_VEL
LIN {X 0,Y 425.354,Z 592.501,A -85,B 0,C 180,E1 -9705.65,E2 -9705.65} C_VEL
LIN {X 0,Y 425.355,Z 592.498,A -85,B 0,C 180,E1 -9708.564,E2 -9708.564} C_VEL
LIN {X 0,Y 425.544,Z 592.476,A -85,B 0,C 180,E1 -9712.408,E2 -9712.408} C_VEL
LIN {X 0,Y 425.557,Z 592.476,A -85,B 0,C 180,E1 -9714.313,E2 -9714.313} C_VEL
LIN {X 0,Y 425.578,Z 592.476,A -85,B 0,C 180,E1 -9718.107,E2 -9718.107} C_VEL
LIN {X 0,Y 425.707,Z 592.458,A -85,B 0,C 180,E1 -9720,E2 -9720} C_VEL
LIN {X 0,Y 425.551,Z 592.473,A -85,B 0,C 180,E1 -9722.84,E2 -9722.84} C_VEL
LIN {X 0,Y 425.535,Z 592.477,A -85,B 0,C 180,E1 -9726.639,E2 -9726.639} C_VEL
LIN {X 0,Y 425.406,Z 592.49,A -85,B 0,C 180,E1 -9729.509,E2 -9729.509} C_VEL
LIN {X 0,Y 425.399,Z 592.493,A -85,B 0,C 180,E1 -9732.904,E2 -9732.904} C_VEL
LIN {X 0,Y 425.367,Z 592.501,A -85,B 0,C 180,E1 -9736.605,E2 -9736.605} C_VEL
LIN {X 0,Y 425.334,Z 592.499,A -85,B 0,C 180,E1 -9739.635,E2 -9739.635} C_VEL
LIN {X 0,Y 425.294,Z 592.508,A -85,B 0,C 180,E1 -9742.339,E2 -9742.339} C_VEL
LIN {X 0,Y 425.298,Z 592.504,A -85,B 0,C 180,E1 -9745.445,E2 -9745.445} C_VEL
LIN {X 0,Y 425.337,Z 592.505,A -85,B 0,C 180,E1 -9748.632,E2 -9748.632} C_VEL
LIN {X 0,Y 425.27,Z 592.507,A -85,B 0,C 180,E1 -9751.927,E2 -9751.927} C_VEL
LIN {X 0,Y 425.305,Z 592.504,A -85,B 0,C 180,E1 -9755.336,E2 -9755.336} C_VEL
LIN {X 0,Y 425.307,Z 592.51,A -85,B 0,C 180,E1 -9758.898,E2 -9758.898} C_VEL
LIN {X 0,Y 425.296,Z 592.504,A -85,B 0,C 180,E1 -9761.958,E2 -9761.958} C_VEL
LIN {X 0,Y 425.29,Z 592.509,A -85,B 0,C 180,E1 -9765.283,E2 -9765.283} C_VEL
LIN {X 0,Y 425.28,Z 592.508,A -85,B 0,C 180,E1 -9768.621,E2 -9768.621} C_VEL
LIN {X 0,Y 425.311,Z 592.51,A -85,B 0,C 180,E1 -9771.102,E2 -9771.102} C_VEL
LIN {X 0,Y 425.305,Z 592.504,A -85,B 0,C 180,E1 -9774.664,E2 -9774.664} C_VEL
LIN {X 0,Y 425.27,Z 592.509,A -85,B 0,C 180,E1 -9778.073,E2 -9778.073} C_VEL
LIN {X 0,Y 425.37,Z 592.629,A -85,B 0,C 180,E1 -9781.3,E2 -9781.3} C_VEL
LIN {X 0,Y 428.075,Z 605.487,A -85,B 0,C 180,E1 -9783.918,E2 -9783.918} C_VEL
LIN {X 0,Y 428.749,Z 609.842,A -85,B 0,C 180,E1 -9784.773,E2 -9784.773} C_VEL
LIN {X 0,Y 428.062,Z 621.762,A -85,B 0,C 180,E1 -9786.965,E2 -9786.965} C_VEL
LIN {X 0,Y 426.965,Z 640.045,A -85,B 0,C 180,E1 -9790.278,E2 -9790.278} C_VEL
LIN {X 0,Y 426.669,Z 646.155,A -85,B 0,C 180,E1 -9791.343,E2 -9791.343} C_VEL
LIN {X 0,Y 430.259,Z 672.256,A -85,B 0,C 180,E1 -9791.973,E2 -9791.973} C_VEL
LIN {X 0,Y 429.217,Z 755.336,A -85,B 0,C 180,E1 -9793.47,E2 -9793.47} C_VEL
LIN {X 0,Y 428.709,Z 768.943,A -85,B 0,C 180,E1 -9793.909,E2 -9793.909} C_VEL
LIN {X 0,Y 428.195,Z 780.767,A -85,B 0,C 180,E1 -9794.469,E2 -9794.469} C_VEL
LIN {X 0,Y 427.455,Z 792.801,A -85,B 0,C 180,E1 -9795.235,E2 -9795.235} C_VEL
LIN {X 0,Y 426.797,Z 804.017,A -85,B 0,C 180,E1 -9796.155,E2 -9796.155} C_VEL
LIN {X 0,Y 426.12,Z 814.758,A -85,B 0,C 180,E1 -9797.255,E2 -9797.255} C_VEL
LIN {X 0,Y 425.608,Z 823.279,A -85,B 0,C 180,E1 -9798.329,E2 -9798.329} C_VEL
LIN {X 0,Y 424.979,Z 832.506,A -85,B 0,C 180,E1 -9799.759,E2 -9799.759} C_VEL
LIN {X 0,Y 424.654,Z 839.946,A -85,B 0,C 180,E1 -9801.193,E2 -9801.193} C_VEL
LIN {X 0,Y 424.387,Z 844.978,A -85,B 0,C 180,E1 -9802.386,E2 -9802.386} C_VEL
LIN {X 0,Y 424.279,Z 849.373,A -85,B 0,C 180,E1 -9803.657,E2 -9803.657} C_VEL
LIN {X 0,Y 424.219,Z 853.594,A -85,B 0,C 180,E1 -9805.247,E2 -9805.247} C_VEL
LIN {X 0,Y 424.142,Z 855.511,A -85,B 0,C 180,E1 -9806.199,E2 -9806.199} C_VEL
LIN {X 0,Y 424.245,Z 856.975,A -85,B 0,C 180,E1 -9807.15,E2 -9807.15} C_VEL
LIN {X 0,Y 424.207,Z 857.993,A -85,B 0,C 180,E1 -9808.1,E2 -9808.1} C_VEL
LIN {X 0,Y 424.19,Z 858.61,A -85,B 0,C 180,E1 -9809.05,E2 -9809.05} C_VEL
LIN {X 0,Y 424.202,Z 858.831,A -85,B 0,C 180,E1 -9809.999,E2 -9809.999} C_VEL
LIN {X 0,Y 424.19,Z 858.608,A -85,B 0,C 180,E1 -9810.948,E2 -9810.948} C_VEL
LIN {X 0,Y 424.209,Z 857.972,A -85,B 0,C 180,E1 -9811.898,E2 -9811.898} C_VEL
LIN {X 0,Y 424.25,Z 856.936,A -85,B 0,C 180,E1 -9812.848,E2 -9812.848} C_VEL
LIN {X 0,Y 424.14,Z 855.481,A -85,B 0,C 180,E1 -9813.799,E2 -9813.799} C_VEL
LIN {X 0,Y 424.237,Z 852.446,A -85,B 0,C 180,E1 -9815.227,E2 -9815.227} C_VEL
LIN {X 0,Y 424.299,Z 848.341,A -85,B 0,C 180,E1 -9816.657,E2 -9816.657} C_VEL
LIN {X 0,Y 424.535,Z 842.037,A -85,B 0,C 180,E1 -9818.328,E2 -9818.328} C_VEL
LIN {X 0,Y 424.878,Z 835.176,A -85,B 0,C 180,E1 -9819.76,E2 -9819.76} C_VEL
LIN {X 0,Y 425.388,Z 826.679,A -85,B 0,C 180,E1 -9821.193,E2 -9821.193} C_VEL
LIN {X 0,Y 425.922,Z 817.947,A -85,B 0,C 180,E1 -9822.386,E2 -9822.386} C_VEL
LIN {X 0,Y 426.55,Z 808.149,A -85,B 0,C 180,E1 -9823.481,E2 -9823.481} C_VEL
LIN {X 0,Y 427.296,Z 796.574,A -85,B 0,C 180,E1 -9824.525,E2 -9824.525} C_VEL
LIN {X 0,Y 428.013,Z 784.853,A -85,B 0,C 180,E1 -9825.352,E2 -9825.352} C_VEL
LIN {X 0,Y 428.581,Z 772.742,A -85,B 0,C 180,E1 -9826.002,E2 -9826.002} C_VEL
LIN {X 0,Y 429.216,Z 759.727,A -85,B 0,C 180,E1 -9826.497,E2 -9826.497} C_VEL
LIN {X 0,Y 429.562,Z 745.933,A -85,B 0,C 180,E1 -9826.82,E2 -9826.82} C_VEL
LIN {X 0,Y 430.418,Z 670.793,A -85,B 0,C 180,E1 -9828.176,E2 -9828.176} C_VEL
LIN {X 0,Y 426.654,Z 644.318,A -85,B 0,C 180,E1 -9828.874,E2 -9828.874} C_VEL
LIN {X 0,Y 427.802,Z 624.726,A -85,B 0,C 180,E1 -9832.442,E2 -9832.442} C_VEL
LIN {X 0,Y 428.787,Z 609.786,A -85,B 0,C 180,E1 -9835.222,E2 -9835.222} C_VEL
LIN {X 0,Y 427.025,Z 599.742,A -85,B 0,C 180,E1 -9837.285,E2 -9837.285} C_VEL
LIN {X 0,Y 425.324,Z 592.51,A -85,B 0,C 180,E1 -9838.864,E2 -9838.864} C_VEL
LIN {X 0,Y 425.262,Z 592.516,A -85,B 0,C 180,E1 -9841.926,E2 -9841.926} C_VEL
LIN {X 0,Y 425.298,Z 592.508,A -85,B 0,C 180,E1 -9845.335,E2 -9845.335} C_VEL
LIN {X 0,Y 425.309,Z 592.508,A -85,B 0,C 180,E1 -9849.045,E2 -9849.045} C_VEL
LIN {X 0,Y 425.311,Z 592.509,A -85,B 0,C 180,E1 -9851.961,E2 -9851.961} C_VEL
LIN {X 0,Y 425.308,Z 592.507,A -85,B 0,C 180,E1 -9855.278,E2 -9855.278} C_VEL
LIN {X 0,Y 425.305,Z 592.508,A -85,B 0,C 180,E1 -9858.625,E2 -9858.625} C_VEL
LIN {X 0,Y 425.319,Z 592.503,A -85,B 0,C 180,E1 -9861.103,E2 -9861.103} C_VEL
LIN {X 0,Y 425.294,Z 592.509,A -85,B 0,C 180,E1 -9864.663,E2 -9864.663} C_VEL
LIN {X 0,Y 425.267,Z 592.511,A -85,B 0,C 180,E1 -9868.073,E2 -9868.073} C_VEL
LIN {X 0,Y 425.331,Z 592.496,A -85,B 0,C 180,E1 -9871.368,E2 -9871.368} C_VEL
LIN {X 0,Y 425.289,Z 592.508,A -85,B 0,C 180,E1 -9874.554,E2 -9874.554} C_VEL
LIN {X 0,Y 425.28,Z 592.506,A -85,B 0,C 180,E1 -9877.661,E2 -9877.661} C_VEL
LIN {X 0,Y 425.354,Z 592.502,A -85,B 0,C 180,E1 -9880.703,E2 -9880.703} C_VEL
LIN {X 0,Y 425.38,Z 592.496,A -85,B 0,C 180,E1 -9883.688,E2 -9883.688} C_VEL
LIN {X 0,Y 425.421,Z 592.489,A -85,B 0,C 180,E1 -9887.598,E2 -9887.598} C_VEL
LIN {X 0,Y 425.434,Z 592.489,A -85,B 0,C 180,E1 -9891.45,E2 -9891.45} C_VEL
LIN {X 0,Y 425.546,Z 592.479,A -85,B 0,C 180,E1 -9894.313,E2 -9894.313} C_VEL
LIN {X 0,Y 425.567,Z 592.477,A -85,B 0,C 180,E1 -9898.107,E2 -9898.107} C_VEL
LIN {X 0,Y 425.696,Z 592.46,A -85,B 0,C 180,E1 -9900,E2 -9900} C_VEL
LIN {X 0,Y 425.55,Z 592.477,A -85,B 0,C 180,E1 -9902.84,E2 -9902.84} C_VEL
LIN {X 0,Y 425.571,Z 592.476,A -85,B 0,C 180,E1 -9905.686,E2 -9905.686} C_VEL
LIN {X 0,Y 425.434,Z 592.494,A -85,B 0,C 180,E1 -9908.55,E2 -9908.55} C_VEL
LIN {X 0,Y 425.418,Z 592.498,A -85,B 0,C 180,E1 -9912.401,E2 -9912.401} C_VEL
LIN {X 0,Y 425.356,Z 592.62,A -85,B 0,C 180,E1 -9913.862,E2 -9913.862} C_VEL
LIN {X 0,Y 426.926,Z 601.036,A -85,B 0,C 180,E1 -9916.19,E2 -9916.19} C_VEL
LIN {X 0,Y 428.082,Z 604.879,A -85,B 0,C 180,E1 -9916.359,E2 -9916.359} C_VEL
LIN {X 0,Y 431.064,Z 617.832,A -85,B 0,C 180,E1 -9916.761,E2 -9916.761} C_VEL
LIN {X 0,Y 429.708,Z 707.494,A -85,B 0,C 180,E1 -9918.412,E2 -9918.412} C_VEL
LIN {X 0,Y 429.352,Z 721.222,A -85,B 0,C 180,E1 -9918.865,E2 -9918.865} C_VEL
LIN {X 0,Y 428.898,Z 733.136,A -85,B 0,C 180,E1 -9919.441,E2 -9919.441} C_VEL
LIN {X 0,Y 428.385,Z 744.165,A -85,B 0,C 180,E1 -9920.152,E2 -9920.152} C_VEL
LIN {X 0,Y 427.738,Z 755.629,A -85,B 0,C 180,E1 -9921.1,E2 -9921.1} C_VEL
LIN {X 0,Y 427.049,Z 765.504,A -85,B 0,C 180,E1 -9922.114,E2 -9922.114} C_VEL
LIN {X 0,Y 426.408,Z 774.889,A -85,B 0,C 180,E1 -9923.301,E2 -9923.301} C_VEL
LIN {X 0,Y 425.827,Z 783.015,A -85,B 0,C 180,E1 -9924.569,E2 -9924.569} C_VEL
LIN {X 0,Y 425.338,Z 790.289,A -85,B 0,C 180,E1 -9925.968,E2 -9925.968} C_VEL
LIN {X 0,Y 424.89,Z 796.985,A -85,B 0,C 180,E1 -9927.59,E2 -9927.59} C_VEL
LIN {X 0,Y 424.575,Z 802.094,A -85,B 0,C 180,E1 -9929.229,E2 -9929.229} C_VEL
LIN {X 0,Y 424.341,Z 805.827,A -85,B 0,C 180,E1 -9930.892,E2 -9930.892} C_VEL
LIN {X 0,Y 424.179,Z 807.986,A -85,B 0,C 180,E1 -9932.331,E2 -9932.331} C_VEL
LIN {X 0,Y 424.065,Z 809.328,A -85,B 0,C 180,E1 -9934.043,E2 -9934.043} C_VEL
LIN {X 0,Y 424.089,Z 809.386,A -85,B 0,C 180,E1 -9935.708,E2 -9935.708} C_VEL
LIN {X 0,Y 424.106,Z 808.269,A -85,B 0,C 180,E1 -9937.307,E2 -9937.307} C_VEL
LIN {X 0,Y 424.267,Z 805.773,A -85,B 0,C 180,E1 -9939.011,E2 -9939.011} C_VEL
LIN {X 0,Y 424.458,Z 802.753,A -85,B 0,C 180,E1 -9940.392,E2 -9940.392} C_VEL
LIN {X 0,Y 424.674,Z 798.422,A -85,B 0,C 180,E1 -9941.868,E2 -9941.868} C_VEL
LIN {X 0,Y 424.977,Z 792.954,A -85,B 0,C 180,E1 -9943.313,E2 -9943.313} C_VEL
LIN {X 0,Y 425.463,Z 786.158,A -85,B 0,C 180,E1 -9944.743,E2 -9944.743} C_VEL
LIN {X 0,Y 425.973,Z 777.948,A -85,B 0,C 180,E1 -9946.138,E2 -9946.138} C_VEL
LIN {X 0,Y 426.56,Z 769.161,A -85,B 0,C 180,E1 -9947.342,E2 -9947.342} C_VEL
LIN {X 0,Y 427.268,Z 758.097,A -85,B 0,C 180,E1 -9948.566,E2 -9948.566} C_VEL
LIN {X 0,Y 427.888,Z 747.238,A -85,B 0,C 180,E1 -9949.524,E2 -9949.524} C_VEL
LIN {X 0,Y 428.519,Z 734.879,A -85,B 0,C 180,E1 -9950.369,E2 -9950.369} C_VEL
LIN {X 0,Y 428.959,Z 723.326,A -85,B 0,C 180,E1 -9950.97,E2 -9950.97} C_VEL
LIN {X 0,Y 429.309,Z 711.219,A -85,B 0,C 180,E1 -9951.423,E2 -9951.423} C_VEL
LIN {X 0,Y 429.544,Z 696.514,A -85,B 0,C 180,E1 -9951.753,E2 -9951.753} C_VEL
LIN {X 0,Y 430.477,Z 616.423,A -85,B 0,C 180,E1 -9953.178,E2 -9953.178} C_VEL
LIN {X 0,Y 426.607,Z 599.515,A -85,B 0,C 180,E1 -9953.657,E2 -9953.657} C_VEL
LIN {X 0,Y 425.353,Z 592.504,A -85,B 0,C 180,E1 -9955.48,E2 -9955.48} C_VEL
LIN {X 0,Y 425.281,Z 592.506,A -85,B 0,C 180,E1 -9959.16,E2 -9959.16} C_VEL
LIN {X 0,Y 424.677,Z 592.588,A -85,B 0,C 180,E1 -9959.951,E2 -9959.951} C_VEL
LIN {X 0,Y 421.864,Z 592.932,A -85,B 0,C 180,E1 -9961.236,E2 -9961.236} C_VEL
LIN {X 0,Y 419.436,Z 593.238,A -85,B 0,C 180,E1 -9962.274,E2 -9962.274} C_VEL
LIN {X 0,Y 418.372,Z 593.367,A -85,B 0,C 180,E1 -9963.076,E2 -9963.076} C_VEL
LIN {X 0,Y 418.276,Z 593.378,A -85,B 0,C 180,E1 -9963.348,E2 -9963.348} C_VEL
LIN {X 0,Y 418.286,Z 593.383,A -85,B 0,C 180,E1 -9966.22,E2 -9966.22} C_VEL
LIN {X 0,Y 418.298,Z 593.383,A -85,B 0,C 180,E1 -9970.2,E2 -9970.2} C_VEL
LIN {X 0,Y 418.316,Z 593.373,A -85,B 0,C 180,E1 -9973.406,E2 -9973.406} C_VEL
LIN {X 0,Y 418.355,Z 593.369,A -85,B 0,C 180,E1 -9976.995,E2 -9976.995} C_VEL
LIN {X 0,Y 418.36,Z 593.375,A -85,B 0,C 180,E1 -9980.33,E2 -9980.33} C_VEL
LIN {X 0,Y 418.494,Z 593.351,A -85,B 0,C 180,E1 -9983.25,E2 -9983.25} C_VEL
LIN {X 0,Y 418.341,Z 593.37,A -85,B 0,C 180,E1 -9985.183,E2 -9985.183} C_VEL
LIN {X 0,Y 418.546,Z 593.347,A -85,B 0,C 180,E1 -9988.077,E2 -9988.077} C_VEL
LIN {X 0,Y 418.672,Z 593.33,A -85,B 0,C 180,E1 -9990.001,E2 -9990.001} C_VEL
LIN {X 0,Y 418.512,Z 593.353,A -85,B 0,C 180,E1 -9992.889,E2 -9992.889} C_VEL
LIN {X 0,Y 418.496,Z 593.357,A -85,B 0,C 180,E1 -9996.752,E2 -9996.752} C_VEL
LIN {X 0,Y 418.344,Z 593.37,A -85,B 0,C 180,E1 -9999.672,E2 -9999.672} C_VEL
LIN {X 0,Y 418.349,Z 593.374,A -85,B 0,C 180,E1 -10003.002,E2 -10003.002} C_VEL
LIN {X 0,Y 418.316,Z 593.379,A -85,B 0,C 180,E1 -10006.736,E2 -10006.736} C_VEL
LIN {X 0,Y 418.274,Z 593.378,A -85,B 0,C 180,E1 -10009.791,E2 -10009.791} C_VEL
LIN {X 0,Y 418.241,Z 593.387,A -85,B 0,C 180,E1 -10012.737,E2 -10012.737} C_VEL
LIN {X 0,Y 418.274,Z 593.378,A -85,B 0,C 180,E1 -10015.905,E2 -10015.905} C_VEL
LIN {X 0,Y 418.268,Z 593.386,A -85,B 0,C 180,E1 -10019.163,E2 -10019.163} C_VEL
LIN {X 0,Y 418.261,Z 593.384,A -85,B 0,C 180,E1 -10022.845,E2 -10022.845} C_VEL
LIN {X 0,Y 418.249,Z 593.381,A -85,B 0,C 180,E1 -10026.239,E2 -10026.239} C_VEL
LIN {X 0,Y 418.255,Z 593.383,A -85,B 0,C 180,E1 -10029.683,E2 -10029.683} C_VEL
LIN {X 0,Y 418.233,Z 593.383,A -85,B 0,C 180,E1 -10032.322,E2 -10032.322} C_VEL
LIN {X 0,Y 418.24,Z 593.387,A -85,B 0,C 180,E1 -10035.109,E2 -10035.109} C_VEL
LIN {X 0,Y 418.244,Z 593.385,A -85,B 0,C 180,E1 -10037.767,E2 -10037.767} C_VEL
LIN {X 0,Y 418.249,Z 593.381,A -85,B 0,C 180,E1 -10040.621,E2 -10040.621} C_VEL
LIN {X 0,Y 418.247,Z 593.384,A -85,B 0,C 180,E1 -10043.976,E2 -10043.976} C_VEL
LIN {X 0,Y 418.262,Z 593.382,A -85,B 0,C 180,E1 -10047.157,E2 -10047.157} C_VEL
LIN {X 0,Y 418.273,Z 593.379,A -85,B 0,C 180,E1 -10050.896,E2 -10050.896} C_VEL
LIN {X 0,Y 418.273,Z 593.382,A -85,B 0,C 180,E1 -10054.096,E2 -10054.096} C_VEL
LIN {X 0,Y 418.237,Z 593.385,A -85,B 0,C 180,E1 -10057.264,E2 -10057.264} C_VEL
LIN {X 0,Y 418.288,Z 593.378,A -85,B 0,C 180,E1 -10060.365,E2 -10060.365} C_VEL
LIN {X 0,Y 418.322,Z 593.375,A -85,B 0,C 180,E1 -10063.405,E2 -10063.405} C_VEL
LIN {X 0,Y 418.352,Z 593.369,A -85,B 0,C 180,E1 -10067,E2 -10067} C_VEL
LIN {X 0,Y 418.345,Z 593.373,A -85,B 0,C 180,E1 -10070.329,E2 -10070.329} C_VEL
LIN {X 0,Y 418.494,Z 593.351,A -85,B 0,C 180,E1 -10073.249,E2 -10073.249} C_VEL
LIN {X 0,Y 418.343,Z 593.37,A -85,B 0,C 180,E1 -10075.182,E2 -10075.182} C_VEL
LIN {X 0,Y 418.548,Z 593.351,A -85,B 0,C 180,E1 -10078.076,E2 -10078.076} C_VEL
LIN {X 0,Y 418.676,Z 593.333,A -85,B 0,C 180,E1 -10080,E2 -10080} C_VEL
LIN {X 0,Y 418.506,Z 593.35,A -85,B 0,C 180,E1 -10082.888,E2 -10082.888} C_VEL
LIN {X 0,Y 418.498,Z 593.353,A -85,B 0,C 180,E1 -10086.751,E2 -10086.751} C_VEL
LIN {X 0,Y 418.346,Z 593.37,A -85,B 0,C 180,E1 -10089.671,E2 -10089.671} C_VEL
LIN {X 0,Y 418.352,Z 593.37,A -85,B 0,C 180,E1 -10093.001,E2 -10093.001} C_VEL
LIN {X 0,Y 418.318,Z 593.378,A -85,B 0,C 180,E1 -10096.735,E2 -10096.735} C_VEL
LIN {X 0,Y 418.276,Z 593.378,A -85,B 0,C 180,E1 -10099.79,E2 -10099.79} C_VEL
LIN {X 0,Y 418.238,Z 593.389,A -85,B 0,C 180,E1 -10102.736,E2 -10102.736} C_VEL
LIN {X 0,Y 418.275,Z 593.379,A -85,B 0,C 180,E1 -10105.904,E2 -10105.904} C_VEL
LIN {X 0,Y 418.271,Z 593.381,A -85,B 0,C 180,E1 -10109.162,E2 -10109.162} C_VEL
LIN {X 0,Y 418.263,Z 593.387,A -85,B 0,C 180,E1 -10112.844,E2 -10112.844} C_VEL
LIN {X 0,Y 418.251,Z 593.382,A -85,B 0,C 180,E1 -10116.238,E2 -10116.238} C_VEL
LIN {X 0,Y 418.252,Z 593.381,A -85,B 0,C 180,E1 -10119.682,E2 -10119.682} C_VEL
LIN {X 0,Y 418.235,Z 593.384,A -85,B 0,C 180,E1 -10122.321,E2 -10122.321} C_VEL
LIN {X 0,Y 418.242,Z 593.389,A -85,B 0,C 180,E1 -10125.108,E2 -10125.108} C_VEL
LIN {X 0,Y 418.246,Z 593.383,A -85,B 0,C 180,E1 -10127.766,E2 -10127.766} C_VEL
LIN {X 0,Y 418.258,Z 593.382,A -85,B 0,C 180,E1 -10130.619,E2 -10130.619} C_VEL
LIN {X 0,Y 418.248,Z 593.382,A -85,B 0,C 180,E1 -10133.975,E2 -10133.975} C_VEL
LIN {X 0,Y 418.263,Z 593.387,A -85,B 0,C 180,E1 -10137.155,E2 -10137.155} C_VEL
LIN {X 0,Y 418.274,Z 593.384,A -85,B 0,C 180,E1 -10140.895,E2 -10140.895} C_VEL
LIN {X 0,Y 418.322,Z 593.632,A -85,B 0,C 180,E1 -10141.067,E2 -10141.067} C_VEL
LIN {X 0,Y 421.094,Z 606.537,A -85,B 0,C 180,E1 -10143.75,E2 -10143.75} C_VEL
LIN {X 0,Y 421.846,Z 612.123,A -85,B 0,C 180,E1 -10144.859,E2 -10144.859} C_VEL
LIN {X 0,Y 420.693,Z 628.592,A -85,B 0,C 180,E1 -10147.92,E2 -10147.92} C_VEL
LIN {X 0,Y 419.758,Z 643.667,A -85,B 0,C 180,E1 -10150.69,E2 -10150.69} C_VEL
LIN {X 0,Y 419.65,Z 645.547,A -85,B 0,C 180,E1 -10151.034,E2 -10151.034} C_VEL
LIN {X 0,Y 423.466,Z 672.764,A -85,B 0,C 180,E1 -10151.71,E2 -10151.71} C_VEL
LIN {X 0,Y 422.344,Z 754.998,A -85,B 0,C 180,E1 -10153.224,E2 -10153.224} C_VEL
LIN {X 0,Y 421.846,Z 768.585,A -85,B 0,C 180,E1 -10153.671,E2 -10153.671} C_VEL
LIN {X 0,Y 421.26,Z 780.943,A -85,B 0,C 180,E1 -10154.269,E2 -10154.269} C_VEL
LIN {X 0,Y 420.432,Z 793.623,A -85,B 0,C 180,E1 -10155.106,E2 -10155.106} C_VEL
LIN {X 0,Y 419.707,Z 805.573,A -85,B 0,C 180,E1 -10156.13,E2 -10156.13} C_VEL
LIN {X 0,Y 419.082,Z 815.162,A -85,B 0,C 180,E1 -10157.161,E2 -10157.161} C_VEL
LIN {X 0,Y 418.49,Z 824.375,A -85,B 0,C 180,E1 -10158.373,E2 -10158.373} C_VEL
LIN {X 0,Y 417.88,Z 833.355,A -85,B 0,C 180,E1 -10159.828,E2 -10159.828} C_VEL
LIN {X 0,Y 417.536,Z 840.554,A -85,B 0,C 180,E1 -10161.286,E2 -10161.286} C_VEL
LIN {X 0,Y 417.266,Z 846.28,A -85,B 0,C 180,E1 -10162.742,E2 -10162.742} C_VEL
LIN {X 0,Y 417.128,Z 850.777,A -85,B 0,C 180,E1 -10164.197,E2 -10164.197} C_VEL
LIN {X 0,Y 417.149,Z 853.149,A -85,B 0,C 180,E1 -10165.167,E2 -10165.167} C_VEL
LIN {X 0,Y 417.054,Z 855.072,A -85,B 0,C 180,E1 -10166.134,E2 -10166.134} C_VEL
LIN {X 0,Y 417.155,Z 856.547,A -85,B 0,C 180,E1 -10167.102,E2 -10167.102} C_VEL
LIN {X 0,Y 417.132,Z 857.57,A -85,B 0,C 180,E1 -10168.068,E2 -10168.068} C_VEL
LIN {X 0,Y 417.107,Z 858.191,A -85,B 0,C 180,E1 -10169.034,E2 -10169.034} C_VEL
LIN {X 0,Y 417.116,Z 858.415,A -85,B 0,C 180,E1 -10169.999,E2 -10169.999} C_VEL
LIN {X 0,Y 417.107,Z 858.198,A -85,B 0,C 180,E1 -10170.964,E2 -10170.964} C_VEL
LIN {X 0,Y 417.133,Z 857.563,A -85,B 0,C 180,E1 -10171.93,E2 -10171.93} C_VEL
LIN {X 0,Y 417.159,Z 856.527,A -85,B 0,C 180,E1 -10172.896,E2 -10172.896} C_VEL
LIN {X 0,Y 417.053,Z 855.076,A -85,B 0,C 180,E1 -10173.864,E2 -10173.864} C_VEL
LIN {X 0,Y 417.148,Z 852.044,A -85,B 0,C 180,E1 -10175.316,E2 -10175.316} C_VEL
LIN {X 0,Y 417.231,Z 847.947,A -85,B 0,C 180,E1 -10176.77,E2 -10176.77} C_VEL
LIN {X 0,Y 417.481,Z 841.66,A -85,B 0,C 180,E1 -10178.469,E2 -10178.469} C_VEL
LIN {X 0,Y 417.85,Z 834.803,A -85,B 0,C 180,E1 -10179.926,E2 -10179.926} C_VEL
LIN {X 0,Y 418.383,Z 826.307,A -85,B 0,C 180,E1 -10181.382,E2 -10181.382} C_VEL
LIN {X 0,Y 418.928,Z 817.586,A -85,B 0,C 180,E1 -10182.596,E2 -10182.596} C_VEL
LIN {X 0,Y 419.657,Z 807.356,A -85,B 0,C 180,E1 -10183.753,E2 -10183.753} C_VEL
LIN {X 0,Y 420.394,Z 796.235,A -85,B 0,C 180,E1 -10184.769,E2 -10184.769} C_VEL
LIN {X 0,Y 421.179,Z 784.556,A -85,B 0,C 180,E1 -10185.608,E2 -10185.608} C_VEL
LIN {X 0,Y 421.846,Z 771.2,A -85,B 0,C 180,E1 -10186.327,E2 -10186.327} C_VEL
LIN {X 0,Y 422.513,Z 757.716,A -85,B 0,C 180,E1 -10186.829,E2 -10186.829} C_VEL
LIN {X 0,Y 422.813,Z 741.231,A -85,B 0,C 180,E1 -10187.19,E2 -10187.19} C_VEL
LIN {X 0,Y 423.711,Z 671.471,A -85,B 0,C 180,E1 -10188.481,E2 -10188.481} C_VEL
LIN {X 0,Y 419.898,Z 645.061,A -85,B 0,C 180,E1 -10189.189,E2 -10189.189} C_VEL
LIN {X 0,Y 419.725,Z 643.739,A -85,B 0,C 180,E1 -10189.25,E2 -10189.25} C_VEL
LIN {X 0,Y 420.948,Z 624.708,A -85,B 0,C 180,E1 -10192.788,E2 -10192.788} C_VEL
LIN {X 0,Y 421.86,Z 610.948,A -85,B 0,C 180,E1 -10195.402,E2 -10195.402} C_VEL
LIN {X 0,Y 419.88,Z 600.293,A -85,B 0,C 180,E1 -10197.652,E2 -10197.652} C_VEL
LIN {X 0,Y 418.271,Z 593.385,A -85,B 0,C 180,E1 -10199.229,E2 -10199.229} C_VEL
LIN {X 0,Y 418.255,Z 593.389,A -85,B 0,C 180,E1 -10202.843,E2 -10202.843} C_VEL
LIN {X 0,Y 418.246,Z 593.388,A -85,B 0,C 180,E1 -10206.238,E2 -10206.238} C_VEL
LIN {X 0,Y 418.261,Z 593.385,A -85,B 0,C 180,E1 -10209.679,E2 -10209.679} C_VEL
LIN {X 0,Y 418.241,Z 593.391,A -85,B 0,C 180,E1 -10212.322,E2 -10212.322} C_VEL
LIN {X 0,Y 418.253,Z 593.386,A -85,B 0,C 180,E1 -10215.111,E2 -10215.111} C_VEL
LIN {X 0,Y 418.287,Z 593.381,A -85,B 0,C 180,E1 -10217.772,E2 -10217.772} C_VEL
LIN {X 0,Y 418.261,Z 593.381,A -85,B 0,C 180,E1 -10221.559,E2 -10221.559} C_VEL
LIN {X 0,Y 418.253,Z 593.382,A -85,B 0,C 180,E1 -10225.158,E2 -10225.158} C_VEL
LIN {X 0,Y 418.243,Z 593.383,A -85,B 0,C 180,E1 -10227.471,E2 -10227.471} C_VEL
LIN {X 0,Y 418.27,Z 593.378,A -85,B 0,C 180,E1 -10230.892,E2 -10230.892} C_VEL
LIN {X 0,Y 418.264,Z 593.381,A -85,B 0,C 180,E1 -10234.095,E2 -10234.095} C_VEL
LIN {X 0,Y 418.23,Z 593.384,A -85,B 0,C 180,E1 -10237.263,E2 -10237.263} C_VEL
LIN {X 0,Y 418.275,Z 593.383,A -85,B 0,C 180,E1 -10240.364,E2 -10240.364} C_VEL
LIN {X 0,Y 418.309,Z 593.376,A -85,B 0,C 180,E1 -10243.404,E2 -10243.404} C_VEL
LIN {X 0,Y 418.347,Z 593.371,A -85,B 0,C 180,E1 -10246.993,E2 -10246.993} C_VEL
LIN {X 0,Y 418.351,Z 593.373,A -85,B 0,C 180,E1 -10250.329,E2 -10250.329} C_VEL
LIN {X 0,Y 418.485,Z 593.354,A -85,B 0,C 180,E1 -10253.249,E2 -10253.249} C_VEL
LIN {X 0,Y 418.334,Z 593.373,A -85,B 0,C 180,E1 -10255.181,E2 -10255.181} C_VEL
LIN {X 0,Y 418.536,Z 593.352,A -85,B 0,C 180,E1 -10258.075,E2 -10258.075} C_VEL
LIN {X 0,Y 418.666,Z 593.336,A -85,B 0,C 180,E1 -10260,E2 -10260} C_VEL
LIN {X 0,Y 418.504,Z 593.355,A -85,B 0,C 180,E1 -10262.888,E2 -10262.888} C_VEL
LIN {X 0,Y 418.486,Z 593.359,A -85,B 0,C 180,E1 -10266.608,E2 -10266.608} C_VEL
LIN {X 0,Y 418.392,Z 593.371,A -85,B 0,C 180,E1 -10268.695,E2 -10268.695} C_VEL
LIN {X 0,Y 418.323,Z 593.377,A -85,B 0,C 180,E1 -10271.631,E2 -10271.631} C_VEL
LIN {X 0,Y 418.329,Z 593.493,A -85,B 0,C 180,E1 -10273.555,E2 -10273.555} C_VEL
